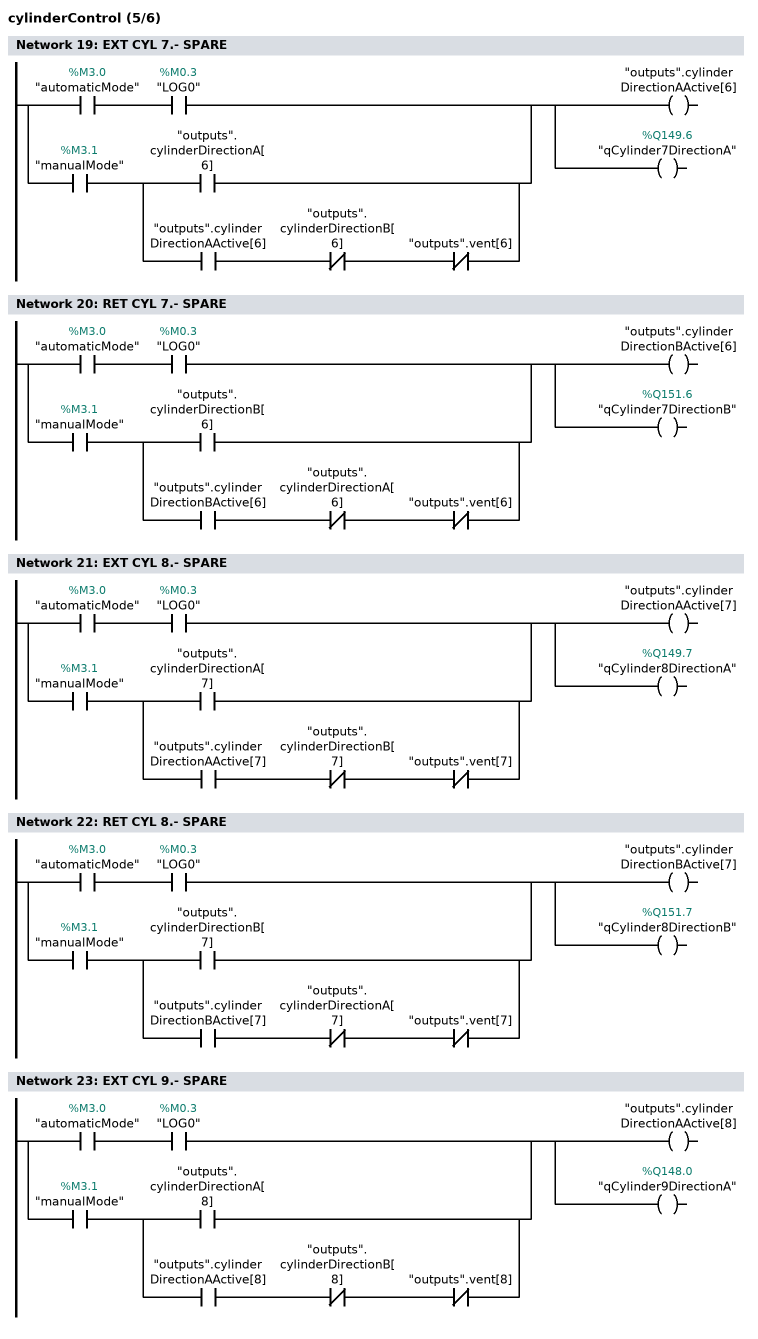
   RUNG wire#powerrail
      Contact( "automaticMode" )
      Contact( "LOG0" )
      wire#w1
      Coil( "outputs".cylinderDirectionAActive[6] )
   END_RUNG
   RUNG wire#powerrail
      Contact( "manualMode" )
      wire#w2
      Contact( "outputs".cylinderDirectionA[6] )
   END_RUNG wire#w1
   RUNG wire#w2
      Contact( "outputs".cylinderDirectionAActive[6] )
      I_Contact( "outputs".cylinderDirectionB[6] )
      I_Contact( "outputs".vent[6] )
   END_RUNG wire#w1
   RUNG wire#w1
      Coil( "qCylinder7DirectionA" )
   END_RUNG
   // the same network as SCL:
   #_w1 := ("automaticMode" AND "LOG0") OR ("manualMode" AND ("outputs".cylinderDirectionA[6] OR ("outputs".cylinderDirectionAActive[6] AND NOT "outputs".cylinderDirectionB[6] AND NOT "outputs".vent[6])));
   "outputs".cylinderDirectionAActive[6] := ("automaticMode" AND "LOG0") OR ("manualMode" AND ("outputs".cylinderDirectionA[6] OR ("outputs".cylinderDirectionAActive[6] AND NOT "outputs".cylinderDirectionB[6] AND NOT "outputs".vent[6])));
   "qCylinder7DirectionA" := #_w1;
END_REGION

REGION Network 20: RET CYL 7.- SPARE
   RUNG wire#powerrail
      Contact( "automaticMode" )
      Contact( "LOG0" )
      wire#w1
      Coil( "outputs".cylinderDirectionBActive[6] )
   END_RUNG
   RUNG wire#powerrail
      Contact( "manualMode" )
      wire#w2
      Contact( "outputs".cylinderDirectionB[6] )
   END_RUNG wire#w1
   RUNG wire#w2
      Contact( "outputs".cylinderDirectionBActive[6] )
      I_Contact( "outputs".cylinderDirectionA[6] )
      I_Contact( "outputs".vent[6] )
   END_RUNG wire#w1
   RUNG wire#w1
      Coil( "qCylinder7DirectionB" )
   END_RUNG
   // the same network as SCL:
   #_w1 := ("automaticMode" AND "LOG0") OR ("manualMode" AND ("outputs".cylinderDirectionB[6] OR ("outputs".cylinderDirectionBActive[6] AND NOT "outputs".cylinderDirectionA[6] AND NOT "outputs".vent[6])));
   "outputs".cylinderDirectionBActive[6] := ("automaticMode" AND "LOG0") OR ("manualMode" AND ("outputs".cylinderDirectionB[6] OR ("outputs".cylinderDirectionBActive[6] AND NOT "outputs".cylinderDirectionA[6] AND NOT "outputs".vent[6])));
   "qCylinder7DirectionB" := #_w1;
END_REGION

REGION Network 21: EXT CYL 8.- SPARE
   RUNG wire#powerrail
      Contact( "automaticMode" )
      Contact( "LOG0" )
      wire#w1
      Coil( "outputs".cylinderDirectionAActive[7] )
   END_RUNG
   RUNG wire#powerrail
      Contact( "manualMode" )
      wire#w2
      Contact( "outputs".cylinderDirectionA[7] )
   END_RUNG wire#w1
   RUNG wire#w2
      Contact( "outputs".cylinderDirectionAActive[7] )
      I_Contact( "outputs".cylinderDirectionB[7] )
      I_Contact( "outputs".vent[7] )
   END_RUNG wire#w1
   RUNG wire#w1
      Coil( "qCylinder8DirectionA" )
   END_RUNG
   // the same network as SCL:
   #_w1 := ("automaticMode" AND "LOG0") OR ("manualMode" AND ("outputs".cylinderDirectionA[7] OR ("outputs".cylinderDirectionAActive[7] AND NOT "outputs".cylinderDirectionB[7] AND NOT "outputs".vent[7])));
   "outputs".cylinderDirectionAActive[7] := ("automaticMode" AND "LOG0") OR ("manualMode" AND ("outputs".cylinderDirectionA[7] OR ("outputs".cylinderDirectionAActive[7] AND NOT "outputs".cylinderDirectionB[7] AND NOT "outputs".vent[7])));
   "qCylinder8DirectionA" := #_w1;
END_REGION

REGION Network 22: RET CYL 8.- SPARE
   RUNG wire#powerrail
      Contact( "automaticMode" )
      Contact( "LOG0" )
      wire#w1
      Coil( "outputs".cylinderDirectionBActive[7] )
   END_RUNG
   RUNG wire#powerrail
      Contact( "manualMode" )
      wire#w2
      Contact( "outputs".cylinderDirectionB[7] )
   END_RUNG wire#w1
   RUNG wire#w2
      Contact( "outputs".cylinderDirectionBActive[7] )
      I_Contact( "outputs".cylinderDirectionA[7] )
      I_Contact( "outputs".vent[7] )
   END_RUNG wire#w1
   RUNG wire#w1
      Coil( "qCylinder8DirectionB" )
   END_RUNG
   // the same network as SCL:
   #_w1 := ("automaticMode" AND "LOG0") OR ("manualMode" AND ("outputs".cylinderDirectionB[7] OR ("outputs".cylinderDirectionBActive[7] AND NOT "outputs".cylinderDirectionA[7] AND NOT "outputs".vent[7])));
   "outputs".cylinderDirectionBActive[7] := ("automaticMode" AND "LOG0") OR ("manualMode" AND ("outputs".cylinderDirectionB[7] OR ("outputs".cylinderDirectionBActive[7] AND NOT "outputs".cylinderDirectionA[7] AND NOT "outputs".vent[7])));
   "qCylinder8DirectionB" := #_w1;
END_REGION

REGION Network 23: EXT CYL 9.- SPARE
   RUNG wire#powerrail
      Contact( "automaticMode" )
      Contact( "LOG0" )
      wire#w1
      Coil( "outputs".cylinderDirectionAActive[8] )
   END_RUNG
   RUNG wire#powerrail
      Contact( "manualMode" )
      wire#w2
      Contact( "outputs".cylinderDirectionA[8] )
   END_RUNG wire#w1
   RUNG wire#w2
      Contact( "outputs".cylinderDirectionAActive[8] )
      I_Contact( "outputs".cylinderDirectionB[8] )
      I_Contact( "outputs".vent[8] )
   END_RUNG wire#w1
   RUNG wire#w1
      Coil( "qCylinder9DirectionA" )
   END_RUNG
   // the same network as SCL:
   #_w1 := ("automaticMode" AND "LOG0") OR ("manualMode" AND ("outputs".cylinderDirectionA[8] OR ("outputs".cylinderDirectionAActive[8] AND NOT "outputs".cylinderDirectionB[8] AND NOT "outputs".vent[8])));
   "outputs".cylinderDirectionAActive[8] := ("automaticMode" AND "LOG0") OR ("manualMode" AND ("outputs".cylinderDirectionA[8] OR ("outputs".cylinderDirectionAActive[8] AND NOT "outputs".cylinderDirectionB[8] AND NOT "outputs".vent[8])));
   "qCylinder9DirectionA" := #_w1;
END_REGION

REGION Network 24: RET CYL 9.- SPARE
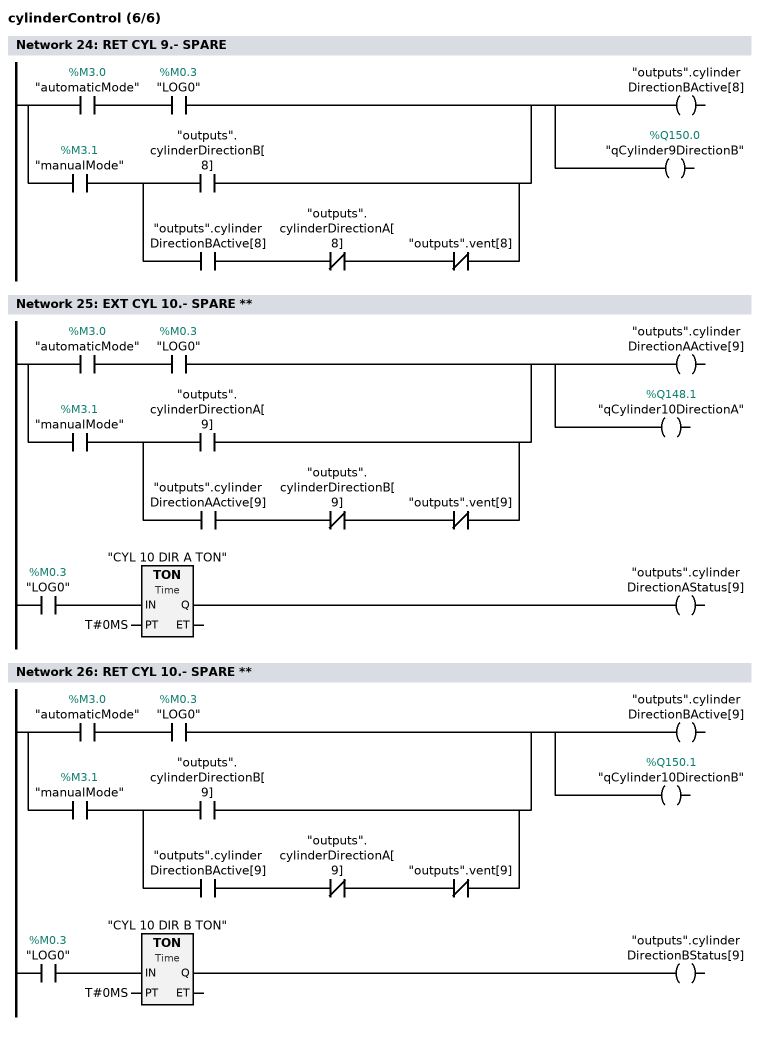
   RUNG wire#powerrail
      Contact( "automaticMode" )
      Contact( "LOG0" )
      wire#w1
      Coil( "outputs".cylinderDirectionBActive[8] )
   END_RUNG
   RUNG wire#powerrail
      Contact( "manualMode" )
      wire#w2
      Contact( "outputs".cylinderDirectionB[8] )
   END_RUNG wire#w1
   RUNG wire#w2
      Contact( "outputs".cylinderDirectionBActive[8] )
      I_Contact( "outputs".cylinderDirectionA[8] )
      I_Contact( "outputs".vent[8] )
   END_RUNG wire#w1
   RUNG wire#w1
      Coil( "qCylinder9DirectionB" )
   END_RUNG
   // the same network as SCL:
   #_w1 := ("automaticMode" AND "LOG0") OR ("manualMode" AND ("outputs".cylinderDirectionB[8] OR ("outputs".cylinderDirectionBActive[8] AND NOT "outputs".cylinderDirectionA[8] AND NOT "outputs".vent[8])));
   "outputs".cylinderDirectionBActive[8] := ("automaticMode" AND "LOG0") OR ("manualMode" AND ("outputs".cylinderDirectionB[8] OR ("outputs".cylinderDirectionBActive[8] AND NOT "outputs".cylinderDirectionA[8] AND NOT "outputs".vent[8])));
   "qCylinder9DirectionB" := #_w1;
END_REGION

REGION Network 25: EXT CYL 10.- SPARE **
   RUNG wire#powerrail
      Contact( "automaticMode" )
      Contact( "LOG0" )
      wire#w1
      Coil( "outputs".cylinderDirectionAActive[9] )
   END_RUNG
   RUNG wire#powerrail
      Contact( "manualMode" )
      wire#w2
      Contact( "outputs".cylinderDirectionA[9] )
   END_RUNG wire#w1
   RUNG wire#w2
      Contact( "outputs".cylinderDirectionAActive[9] )
      I_Contact( "outputs".cylinderDirectionB[9] )
      I_Contact( "outputs".vent[9] )
   END_RUNG wire#w1
   RUNG wire#w1
      Coil( "qCylinder10DirectionA" )
   END_RUNG
   RUNG wire#powerrail
      Contact( "LOG0" )
      { S7_Templates := "time_type := Time" } "CYL 10 DIR A TON".TON(pt := T#0MS, et =>)
      Coil( "outputs".cylinderDirectionAStatus[9] )
   END_RUNG
   // the same network as SCL:
   #_w1 := ("automaticMode" AND "LOG0") OR ("manualMode" AND ("outputs".cylinderDirectionA[9] OR ("outputs".cylinderDirectionAActive[9] AND NOT "outputs".cylinderDirectionB[9] AND NOT "outputs".vent[9])));
   "outputs".cylinderDirectionAActive[9] := ("automaticMode" AND "LOG0") OR ("manualMode" AND ("outputs".cylinderDirectionA[9] OR ("outputs".cylinderDirectionAActive[9] AND NOT "outputs".cylinderDirectionB[9] AND NOT "outputs".vent[9])));
   "qCylinder10DirectionA" := #_w1;
   "CYL 10 DIR A TON".TON(IN := "LOG0", PT := T#0MS);
   "outputs".cylinderDirectionAStatus[9] := "CYL 10 DIR A TON".Q;
END_REGION

REGION Network 26: RET CYL 10.- SPARE **
   RUNG wire#powerrail
      Contact( "automaticMode" )
      Contact( "LOG0" )
      wire#w1
      Coil( "outputs".cylinderDirectionBActive[9] )
   END_RUNG
   RUNG wire#powerrail
      Contact( "manualMode" )
      wire#w2
      Contact( "outputs".cylinderDirectionB[9] )
   END_RUNG wire#w1
   RUNG wire#w2
      Contact( "outputs".cylinderDirectionBActive[9] )
      I_Contact( "outputs".cylinderDirectionA[9] )
      I_Contact( "outputs".vent[9] )
   END_RUNG wire#w1
   RUNG wire#w1
      Coil( "qCylinder10DirectionB" )
   END_RUNG
   RUNG wire#powerrail
      Contact( "LOG0" )
      { S7_Templates := "time_type := Time" } "CYL 10 DIR B TON".TON(pt := T#0MS, et =>)
      Coil( "outputs".cylinderDirectionBStatus[9] )
   END_RUNG
   // the same network as SCL:
   #_w1 := ("automaticMode" AND "LOG0") OR ("manualMode" AND ("outputs".cylinderDirectionB[9] OR ("outputs".cylinderDirectionBActive[9] AND NOT "outputs".cylinderDirectionA[9] AND NOT "outputs".vent[9])));
   "outputs".cylinderDirectionBActive[9] := ("automaticMode" AND "LOG0") OR ("manualMode" AND ("outputs".cylinderDirectionB[9] OR ("outputs".cylinderDirectionBActive[9] AND NOT "outputs".cylinderDirectionA[9] AND NOT "outputs".vent[9])));
   "qCylinder10DirectionB" := #_w1;
   "CYL 10 DIR B TON".TON(IN := "LOG0", PT := T#0MS);
   "outputs".cylinderDirectionBStatus[9] := "CYL 10 DIR B TON".Q;
END_REGION
END_FUNCTION

FUNCTION "outputsMapping" : Void   // FC8, LAD
{ S7_Optimized_Access := 'TRUE' }
VERSION : 0.1
// stored: AutoNumber true, IsIECCheckEnabled false, SetENOAutomatically false, UDAEnableTagReadback false
BEGIN

REGION Network 1: STATION AIR ACTIVATION
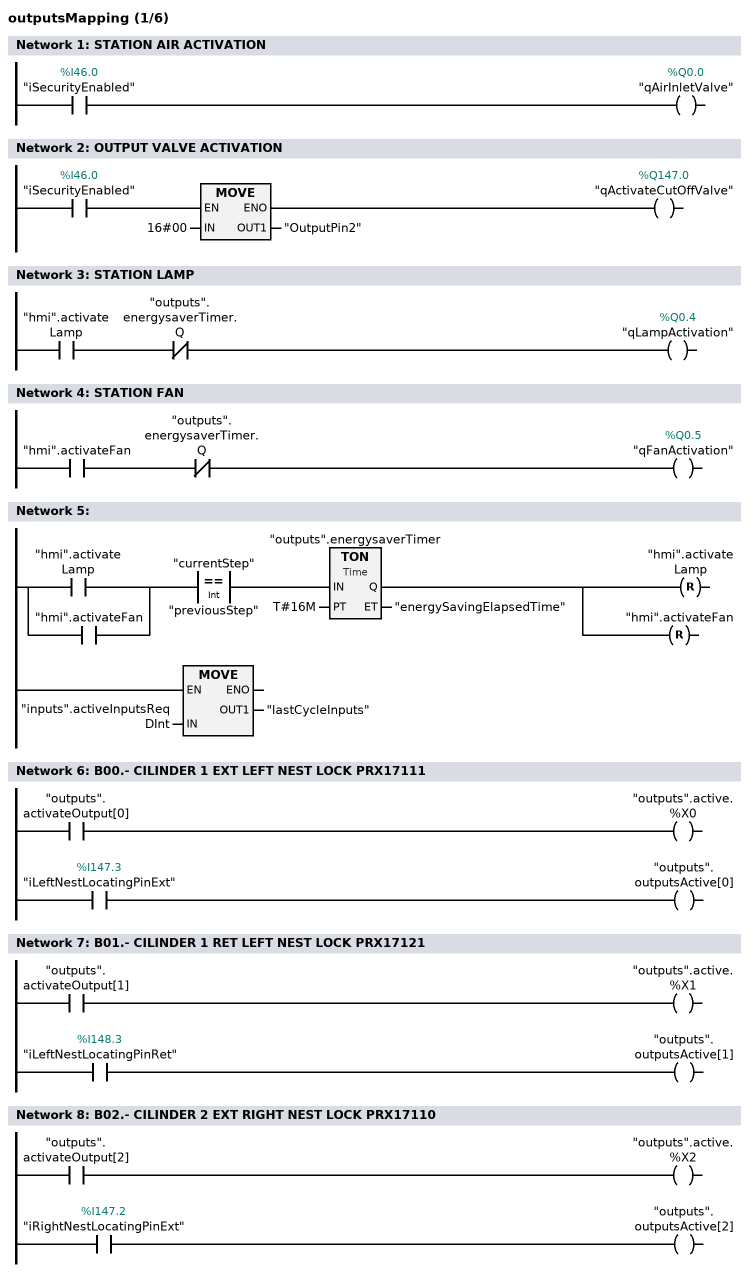
   RUNG wire#powerrail
      Contact( "iSecurityEnabled" )
      Coil( "qAirInletValve" )
   END_RUNG
   // the same network as SCL:
   "qAirInletValve" := "iSecurityEnabled";
END_REGION

REGION Network 2: OUTPUT VALVE ACTIVATION
   RUNG wire#powerrail
      Contact( "iSecurityEnabled" )
      Move(in := 16#00, out1 => "OutputPin2")
      Coil( "qActivateCutOffValve" )
   END_RUNG
   // the same network as SCL:
   IF "iSecurityEnabled" THEN "OutputPin2" := 16#00; END_IF;
   "qActivateCutOffValve" := "iSecurityEnabled";
END_REGION

REGION Network 3: STATION LAMP
   RUNG wire#powerrail
      Contact( "hmi".activateLamp )
      I_Contact( "outputs".energysaverTimer.Q )
      Coil( "qLampActivation" )
   END_RUNG
   // the same network as SCL:
   "qLampActivation" := "hmi".activateLamp AND NOT "outputs".energysaverTimer.Q;
END_REGION

REGION Network 4: STATION FAN
   RUNG wire#powerrail
      Contact( "hmi".activateFan )
      I_Contact( "outputs".energysaverTimer.Q )
      Coil( "qFanActivation" )
   END_RUNG
   // the same network as SCL:
   "qFanActivation" := "hmi".activateFan AND NOT "outputs".energysaverTimer.Q;
END_REGION

REGION Network 5
   RUNG wire#powerrail
      Contact( "hmi".activateLamp )
      wire#w1
      { S7_Templates := "SrcType := Int" } EQ_Contact(in1 := "currentStep", in2 := "previousStep")
      { S7_Templates := "time_type := Time" } "outputs".energysaverTimer.TON(pt := T#16M, et => "energySavingElapsedTime")
      wire#w2
      R_Coil( "hmi".activateLamp )
   END_RUNG
   RUNG wire#powerrail
      Contact( "hmi".activateFan )
   END_RUNG wire#w1
   RUNG wire#w2
      R_Coil( "hmi".activateFan )
   END_RUNG
   RUNG wire#powerrail
      Move(in := "inputs".activeInputsReqDInt, out1 => "lastCycleInputs")
   END_RUNG
   // the same network as SCL:
   "outputs".energysaverTimer.TON(IN := ("hmi".activateLamp OR "hmi".activateFan) AND ("currentStep" = "previousStep"),
                           PT := T#16M,
                           ET => "energySavingElapsedTime");
   IF "outputs".energysaverTimer.Q THEN
       "hmi".activateLamp := FALSE;
       "hmi".activateFan := FALSE;
   END_IF;
   "lastCycleInputs" := "inputs".activeInputsReqDInt;
END_REGION

REGION Network 6: B00.- CILINDER 1 EXT LEFT NEST LOCK PRX17111
   RUNG wire#powerrail
      Contact( "outputs".activateOutput[0] )
      Coil( "outputs".active.%X0 )
   END_RUNG
   RUNG wire#powerrail
      Contact( "iLeftNestLocatingPinExt" )
      Coil( "outputs".outputsActive[0] )
   END_RUNG
   // the same network as SCL:
   "outputs".active.%X0 := "outputs".activateOutput[0];
   "outputs".outputsActive[0] := "iLeftNestLocatingPinExt";
END_REGION

REGION Network 7: B01.- CILINDER 1 RET LEFT NEST LOCK PRX17121
   RUNG wire#powerrail
      Contact( "outputs".activateOutput[1] )
      Coil( "outputs".active.%X1 )
   END_RUNG
   RUNG wire#powerrail
      Contact( "iLeftNestLocatingPinRet" )
      Coil( "outputs".outputsActive[1] )
   END_RUNG
   // the same network as SCL:
   "outputs".active.%X1 := "outputs".activateOutput[1];
   "outputs".outputsActive[1] := "iLeftNestLocatingPinRet";
END_REGION

REGION Network 8: B02.- CILINDER 2 EXT RIGHT NEST LOCK PRX17110
   RUNG wire#powerrail
      Contact( "outputs".activateOutput[2] )
      Coil( "outputs".active.%X2 )
   END_RUNG
   RUNG wire#powerrail
      Contact( "iRightNestLocatingPinExt" )
      Coil( "outputs".outputsActive[2] )
   END_RUNG
   // the same network as SCL:
   "outputs".active.%X2 := "outputs".activateOutput[2];
   "outputs".outputsActive[2] := "iRightNestLocatingPinExt";
END_REGION

REGION Network 9: B03.- CILINDER 2 RET RIGHT NEST LOCK PRX17120
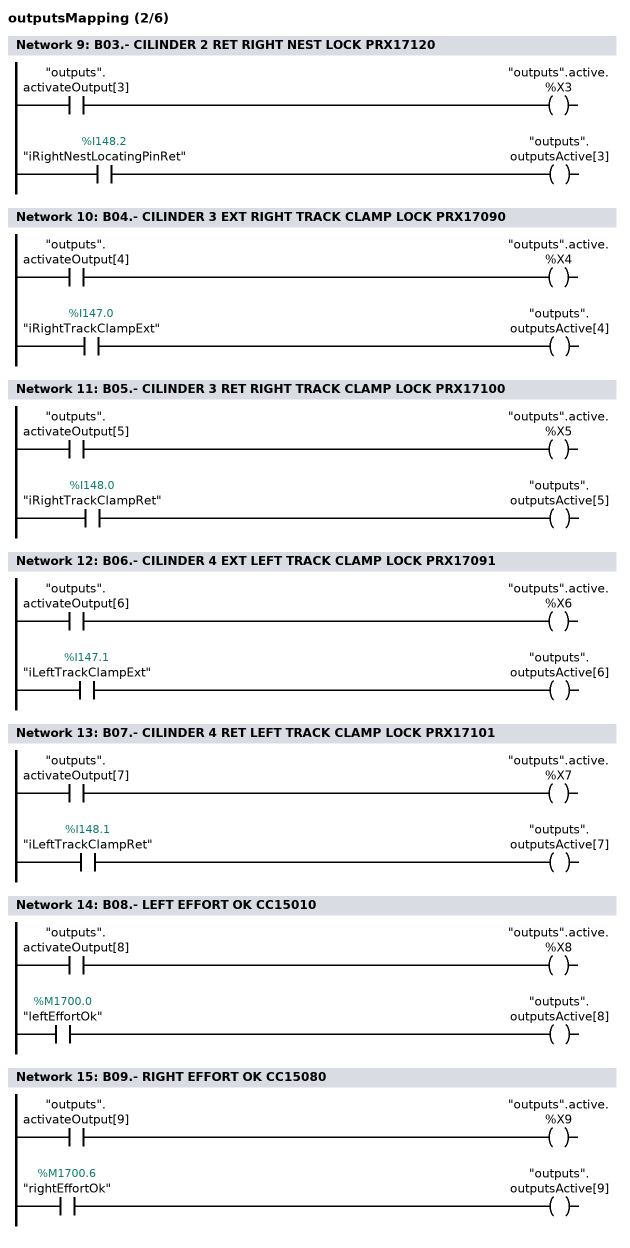
   RUNG wire#powerrail
      Contact( "outputs".activateOutput[3] )
      Coil( "outputs".active.%X3 )
   END_RUNG
   RUNG wire#powerrail
      Contact( "iRightNestLocatingPinRet" )
      Coil( "outputs".outputsActive[3] )
   END_RUNG
   // the same network as SCL:
   "outputs".active.%X3 := "outputs".activateOutput[3];
   "outputs".outputsActive[3] := "iRightNestLocatingPinRet";
END_REGION

REGION Network 10: B04.- CILINDER 3 EXT RIGHT TRACK CLAMP LOCK PRX17090
   RUNG wire#powerrail
      Contact( "outputs".activateOutput[4] )
      Coil( "outputs".active.%X4 )
   END_RUNG
   RUNG wire#powerrail
      Contact( "iRightTrackClampExt" )
      Coil( "outputs".outputsActive[4] )
   END_RUNG
   // the same network as SCL:
   "outputs".active.%X4 := "outputs".activateOutput[4];
   "outputs".outputsActive[4] := "iRightTrackClampExt";
END_REGION

REGION Network 11: B05.- CILINDER 3 RET RIGHT TRACK CLAMP LOCK PRX17100
   RUNG wire#powerrail
      Contact( "outputs".activateOutput[5] )
      Coil( "outputs".active.%X5 )
   END_RUNG
   RUNG wire#powerrail
      Contact( "iRightTrackClampRet" )
      Coil( "outputs".outputsActive[5] )
   END_RUNG
   // the same network as SCL:
   "outputs".active.%X5 := "outputs".activateOutput[5];
   "outputs".outputsActive[5] := "iRightTrackClampRet";
END_REGION

REGION Network 12: B06.- CILINDER 4 EXT LEFT TRACK CLAMP LOCK PRX17091
   RUNG wire#powerrail
      Contact( "outputs".activateOutput[6] )
      Coil( "outputs".active.%X6 )
   END_RUNG
   RUNG wire#powerrail
      Contact( "iLeftTrackClampExt" )
      Coil( "outputs".outputsActive[6] )
   END_RUNG
   // the same network as SCL:
   "outputs".active.%X6 := "outputs".activateOutput[6];
   "outputs".outputsActive[6] := "iLeftTrackClampExt";
END_REGION

REGION Network 13: B07.- CILINDER 4 RET LEFT TRACK CLAMP LOCK PRX17101
   RUNG wire#powerrail
      Contact( "outputs".activateOutput[7] )
      Coil( "outputs".active.%X7 )
   END_RUNG
   RUNG wire#powerrail
      Contact( "iLeftTrackClampRet" )
      Coil( "outputs".outputsActive[7] )
   END_RUNG
   // the same network as SCL:
   "outputs".active.%X7 := "outputs".activateOutput[7];
   "outputs".outputsActive[7] := "iLeftTrackClampRet";
END_REGION

REGION Network 14: B08.- LEFT EFFORT OK CC15010
   RUNG wire#powerrail
      Contact( "outputs".activateOutput[8] )
      Coil( "outputs".active.%X8 )
   END_RUNG
   RUNG wire#powerrail
      Contact( "leftEffortOk" )
      Coil( "outputs".outputsActive[8] )
   END_RUNG
   // the same network as SCL:
   "outputs".active.%X8 := "outputs".activateOutput[8];
   "outputs".outputsActive[8] := "leftEffortOk";
END_REGION

REGION Network 15: B09.- RIGHT EFFORT OK CC15080
   RUNG wire#powerrail
      Contact( "outputs".activateOutput[9] )
      Coil( "outputs".active.%X9 )
   END_RUNG
   RUNG wire#powerrail
      Contact( "rightEffortOk" )
      Coil( "outputs".outputsActive[9] )
   END_RUNG
   // the same network as SCL:
   "outputs".active.%X9 := "outputs".activateOutput[9];
   "outputs".outputsActive[9] := "rightEffortOk";
END_REGION

REGION Network 16: B10.- LEFT INSERTION OK DISTANCE SD14160
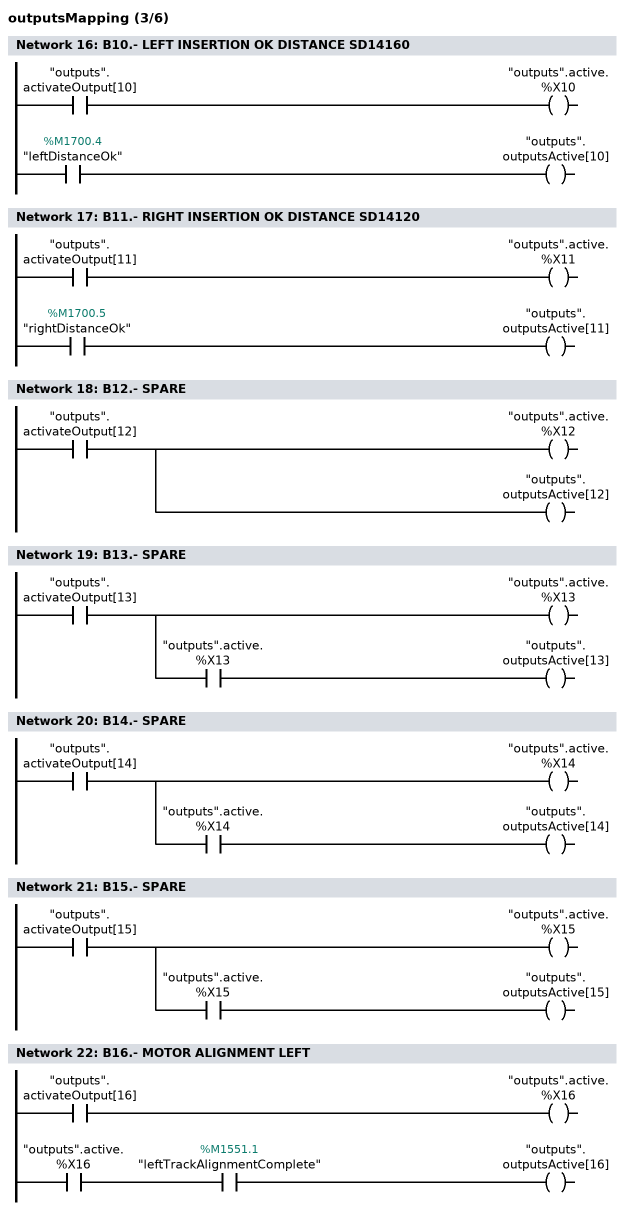
   RUNG wire#powerrail
      Contact( "outputs".activateOutput[10] )
      Coil( "outputs".active.%X10 )
   END_RUNG
   RUNG wire#powerrail
      Contact( "leftDistanceOk" )
      Coil( "outputs".outputsActive[10] )
   END_RUNG
   // the same network as SCL:
   "outputs".active.%X10 := "outputs".activateOutput[10];
   "outputs".outputsActive[10] := "leftDistanceOk";
END_REGION

REGION Network 17: B11.- RIGHT INSERTION OK DISTANCE SD14120
   RUNG wire#powerrail
      Contact( "outputs".activateOutput[11] )
      Coil( "outputs".active.%X11 )
   END_RUNG
   RUNG wire#powerrail
      Contact( "rightDistanceOk" )
      Coil( "outputs".outputsActive[11] )
   END_RUNG
   // the same network as SCL:
   "outputs".active.%X11 := "outputs".activateOutput[11];
   "outputs".outputsActive[11] := "rightDistanceOk";
END_REGION

REGION Network 18: B12.- SPARE
   RUNG wire#powerrail
      Contact( "outputs".activateOutput[12] )
      wire#w1
      Coil( "outputs".active.%X12 )
   END_RUNG
   RUNG wire#w1
      Coil( "outputs".outputsActive[12] )
   END_RUNG
   // the same network as SCL:
   "outputs".active.%X12 := "outputs".activateOutput[12];
   "outputs".outputsActive[12] := "outputs".activateOutput[12];
END_REGION

REGION Network 19: B13.- SPARE
   RUNG wire#powerrail
      Contact( "outputs".activateOutput[13] )
      wire#w1
      Coil( "outputs".active.%X13 )
   END_RUNG
   RUNG wire#w1
      Contact( "outputs".active.%X13 )
      Coil( "outputs".outputsActive[13] )
   END_RUNG
   // the same network as SCL:
   "outputs".active.%X13 := "outputs".activateOutput[13];
   "outputs".outputsActive[13] := "outputs".activateOutput[13] AND "outputs".active.%X13;
END_REGION

REGION Network 20: B14.- SPARE
   RUNG wire#powerrail
      Contact( "outputs".activateOutput[14] )
      wire#w1
      Coil( "outputs".active.%X14 )
   END_RUNG
   RUNG wire#w1
      Contact( "outputs".active.%X14 )
      Coil( "outputs".outputsActive[14] )
   END_RUNG
   // the same network as SCL:
   "outputs".active.%X14 := "outputs".activateOutput[14];
   "outputs".outputsActive[14] := "outputs".activateOutput[14] AND "outputs".active.%X14;
END_REGION

REGION Network 21: B15.- SPARE
   RUNG wire#powerrail
      Contact( "outputs".activateOutput[15] )
      wire#w1
      Coil( "outputs".active.%X15 )
   END_RUNG
   RUNG wire#w1
      Contact( "outputs".active.%X15 )
      Coil( "outputs".outputsActive[15] )
   END_RUNG
   // the same network as SCL:
   "outputs".active.%X15 := "outputs".activateOutput[15];
   "outputs".outputsActive[15] := "outputs".activateOutput[15] AND "outputs".active.%X15;
END_REGION

REGION Network 22: B16.- MOTOR ALIGNMENT LEFT
   RUNG wire#powerrail
      Contact( "outputs".activateOutput[16] )
      Coil( "outputs".active.%X16 )
   END_RUNG
   RUNG wire#powerrail
      Contact( "outputs".active.%X16 )
      Contact( "leftTrackAlignmentComplete" )
      Coil( "outputs".outputsActive[16] )
   END_RUNG
   // the same network as SCL:
   "outputs".active.%X16 := "outputs".activateOutput[16];
   "outputs".outputsActive[16] := "outputs".active.%X16 AND "leftTrackAlignmentComplete";
END_REGION

REGION Network 23: B17.- MOTOR ALIGNMENT RIGHT
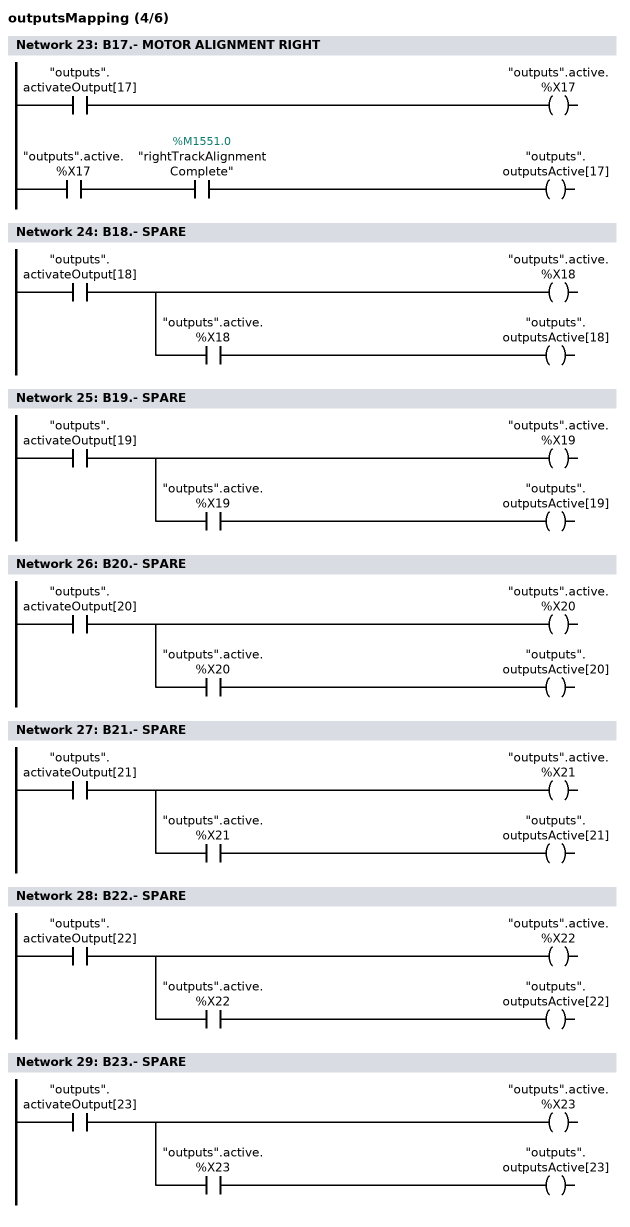
   RUNG wire#powerrail
      Contact( "outputs".activateOutput[17] )
      Coil( "outputs".active.%X17 )
   END_RUNG
   RUNG wire#powerrail
      Contact( "outputs".active.%X17 )
      Contact( "rightTrackAlignmentComplete" )
      Coil( "outputs".outputsActive[17] )
   END_RUNG
   // the same network as SCL:
   "outputs".active.%X17 := "outputs".activateOutput[17];
   "outputs".outputsActive[17] := "outputs".active.%X17 AND "rightTrackAlignmentComplete";
END_REGION

REGION Network 24: B18.- SPARE
   RUNG wire#powerrail
      Contact( "outputs".activateOutput[18] )
      wire#w1
      Coil( "outputs".active.%X18 )
   END_RUNG
   RUNG wire#w1
      Contact( "outputs".active.%X18 )
      Coil( "outputs".outputsActive[18] )
   END_RUNG
   // the same network as SCL:
   "outputs".active.%X18 := "outputs".activateOutput[18];
   "outputs".outputsActive[18] := "outputs".activateOutput[18] AND "outputs".active.%X18;
END_REGION

REGION Network 25: B19.- SPARE
   RUNG wire#powerrail
      Contact( "outputs".activateOutput[19] )
      wire#w1
      Coil( "outputs".active.%X19 )
   END_RUNG
   RUNG wire#w1
      Contact( "outputs".active.%X19 )
      Coil( "outputs".outputsActive[19] )
   END_RUNG
   // the same network as SCL:
   "outputs".active.%X19 := "outputs".activateOutput[19];
   "outputs".outputsActive[19] := "outputs".activateOutput[19] AND "outputs".active.%X19;
END_REGION

REGION Network 26: B20.- SPARE
   RUNG wire#powerrail
      Contact( "outputs".activateOutput[20] )
      wire#w1
      Coil( "outputs".active.%X20 )
   END_RUNG
   RUNG wire#w1
      Contact( "outputs".active.%X20 )
      Coil( "outputs".outputsActive[20] )
   END_RUNG
   // the same network as SCL:
   "outputs".active.%X20 := "outputs".activateOutput[20];
   "outputs".outputsActive[20] := "outputs".activateOutput[20] AND "outputs".active.%X20;
END_REGION

REGION Network 27: B21.- SPARE
   RUNG wire#powerrail
      Contact( "outputs".activateOutput[21] )
      wire#w1
      Coil( "outputs".active.%X21 )
   END_RUNG
   RUNG wire#w1
      Contact( "outputs".active.%X21 )
      Coil( "outputs".outputsActive[21] )
   END_RUNG
   // the same network as SCL:
   "outputs".active.%X21 := "outputs".activateOutput[21];
   "outputs".outputsActive[21] := "outputs".activateOutput[21] AND "outputs".active.%X21;
END_REGION

REGION Network 28: B22.- SPARE
   RUNG wire#powerrail
      Contact( "outputs".activateOutput[22] )
      wire#w1
      Coil( "outputs".active.%X22 )
   END_RUNG
   RUNG wire#w1
      Contact( "outputs".active.%X22 )
      Coil( "outputs".outputsActive[22] )
   END_RUNG
   // the same network as SCL:
   "outputs".active.%X22 := "outputs".activateOutput[22];
   "outputs".outputsActive[22] := "outputs".activateOutput[22] AND "outputs".active.%X22;
END_REGION

REGION Network 29: B23.- SPARE
   RUNG wire#powerrail
      Contact( "outputs".activateOutput[23] )
      wire#w1
      Coil( "outputs".active.%X23 )
   END_RUNG
   RUNG wire#w1
      Contact( "outputs".active.%X23 )
      Coil( "outputs".outputsActive[23] )
   END_RUNG
   // the same network as SCL:
   "outputs".active.%X23 := "outputs".activateOutput[23];
   "outputs".outputsActive[23] := "outputs".activateOutput[23] AND "outputs".active.%X23;
END_REGION

REGION Network 30: B24.- SPARE
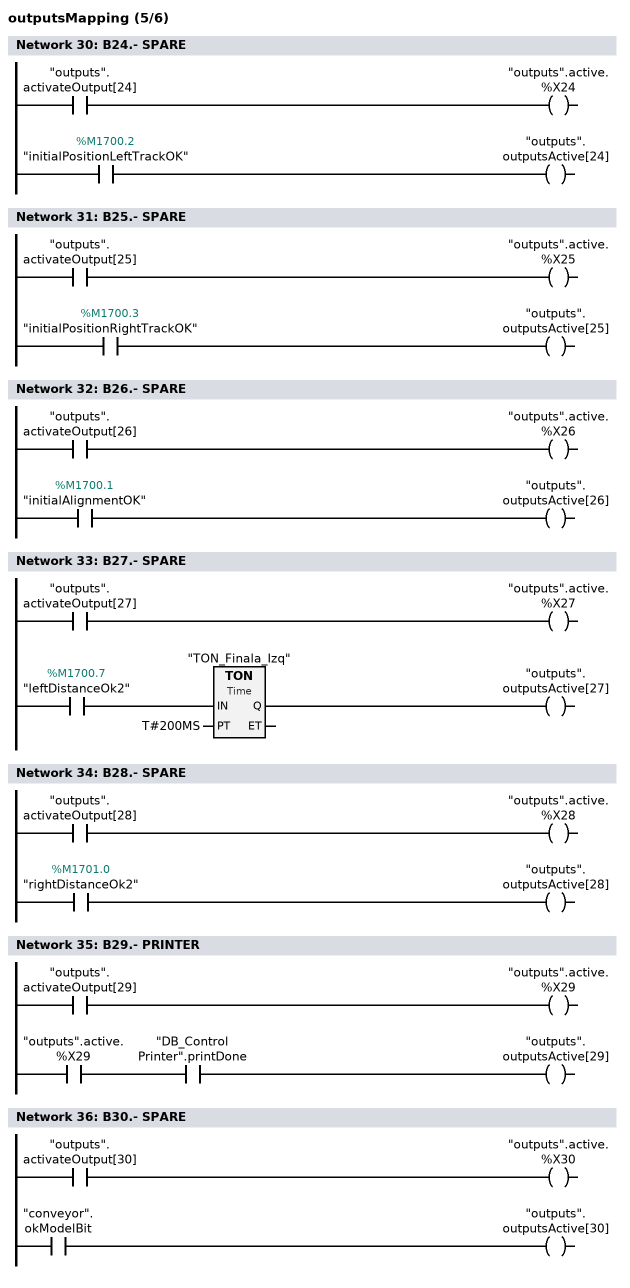
   RUNG wire#powerrail
      Contact( "outputs".activateOutput[24] )
      Coil( "outputs".active.%X24 )
   END_RUNG
   RUNG wire#powerrail
      Contact( "initialPositionLeftTrackOK" )
      Coil( "outputs".outputsActive[24] )
   END_RUNG
   // the same network as SCL:
   "outputs".active.%X24 := "outputs".activateOutput[24];
   "outputs".outputsActive[24] := "initialPositionLeftTrackOK";
END_REGION

REGION Network 31: B25.- SPARE
   RUNG wire#powerrail
      Contact( "outputs".activateOutput[25] )
      Coil( "outputs".active.%X25 )
   END_RUNG
   RUNG wire#powerrail
      Contact( "initialPositionRightTrackOK" )
      Coil( "outputs".outputsActive[25] )
   END_RUNG
   // the same network as SCL:
   "outputs".active.%X25 := "outputs".activateOutput[25];
   "outputs".outputsActive[25] := "initialPositionRightTrackOK";
END_REGION

REGION Network 32: B26.- SPARE
   RUNG wire#powerrail
      Contact( "outputs".activateOutput[26] )
      Coil( "outputs".active.%X26 )
   END_RUNG
   RUNG wire#powerrail
      Contact( "initialAlignmentOK" )
      Coil( "outputs".outputsActive[26] )
   END_RUNG
   // the same network as SCL:
   "outputs".active.%X26 := "outputs".activateOutput[26];
   "outputs".outputsActive[26] := "initialAlignmentOK";
END_REGION

REGION Network 33: B27.- SPARE
   RUNG wire#powerrail
      Contact( "outputs".activateOutput[27] )
      Coil( "outputs".active.%X27 )
   END_RUNG
   RUNG wire#powerrail
      Contact( "leftDistanceOk2" )
      { S7_Templates := "time_type := Time" } "TON_Finala_Izq".TON(pt := T#200MS, et =>)
      Coil( "outputs".outputsActive[27] )
   END_RUNG
   // the same network as SCL:
   "outputs".active.%X27 := "outputs".activateOutput[27];
   "TON_Finala_Izq".TON(IN := "leftDistanceOk2", PT := T#200MS);
   "outputs".outputsActive[27] := "TON_Finala_Izq".Q;
END_REGION

REGION Network 34: B28.- SPARE
   RUNG wire#powerrail
      Contact( "outputs".activateOutput[28] )
      Coil( "outputs".active.%X28 )
   END_RUNG
   RUNG wire#powerrail
      Contact( "rightDistanceOk2" )
      Coil( "outputs".outputsActive[28] )
   END_RUNG
   // the same network as SCL:
   "outputs".active.%X28 := "outputs".activateOutput[28];
   "outputs".outputsActive[28] := "rightDistanceOk2";
END_REGION

REGION Network 35: B29.- PRINTER
   RUNG wire#powerrail
      Contact( "outputs".activateOutput[29] )
      Coil( "outputs".active.%X29 )
   END_RUNG
   RUNG wire#powerrail
      Contact( "outputs".active.%X29 )
      Contact( "DB_ControlPrinter".printDone )
      Coil( "outputs".outputsActive[29] )
   END_RUNG
   // the same network as SCL:
   "outputs".active.%X29 := "outputs".activateOutput[29];
   "outputs".outputsActive[29] := "outputs".active.%X29 AND "DB_ControlPrinter".printDone;
END_REGION

REGION Network 36: B30.- SPARE
   RUNG wire#powerrail
      Contact( "outputs".activateOutput[30] )
      Coil( "outputs".active.%X30 )
   END_RUNG
   RUNG wire#powerrail
      Contact( "conveyor".okModelBit )
      Coil( "outputs".outputsActive[30] )
   END_RUNG
   // the same network as SCL:
   "outputs".active.%X30 := "outputs".activateOutput[30];
   "outputs".outputsActive[30] := "conveyor".okModelBit;
END_REGION

REGION Network 37: B31.- CYCLE TIME
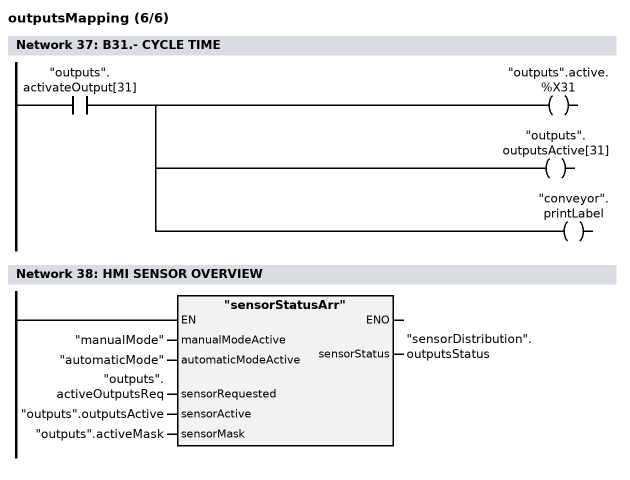
   RUNG wire#powerrail
      Contact( "outputs".activateOutput[31] )
      wire#w1
      Coil( "outputs".active.%X31 )
   END_RUNG
   RUNG wire#w1
      Coil( "outputs".outputsActive[31] )
   END_RUNG
   RUNG wire#w1
      Coil( "conveyor".printLabel )
   END_RUNG
   // the same network as SCL:
   "outputs".active.%X31 := "outputs".activateOutput[31];
   "outputs".outputsActive[31] := "outputs".activateOutput[31];
   "conveyor".printLabel := "outputs".activateOutput[31];
END_REGION

REGION Network 38: HMI SENSOR OVERVIEW
   RUNG wire#powerrail
      "sensorStatusArr"(manualModeActive := "manualMode", automaticModeActive := "automaticMode", sensorRequested := "outputs".activeOutputsReq, sensorActive := "outputs".outputsActive, sensorMask := "outputs".activeMask, sensorStatus => "sensorDistribution".outputsStatus)
   END_RUNG
   // the same network as SCL:
   "sensorStatusArr"(manualModeActive := "manualMode",
                     automaticModeActive := "automaticMode",
                     sensorRequested := "outputs".activeOutputsReq,
                     sensorActive := "outputs".outputsActive,
                     sensorMask := "outputs".activeMask,
                     sensorStatus => "sensorDistribution".outputsStatus);
END_REGION
END_FUNCTION

FUNCTION "sensorStatusArr" : Void   // FC38, LAD
{ S7_Optimized_Access := 'TRUE' }
VERSION : 0.1
// stored: AutoNumber true, IsIECCheckEnabled false, SetENOAutomatically false, UDAEnableTagReadback false
   VAR_INPUT
      manualModeActive : Bool;
      automaticModeActive : Bool;
      sensorRequested : Array[0..31] of Bool;
      sensorActive : Array[0..31] of Bool;
      sensorMask : Array[0..31] of Bool;
   END_VAR
   VAR_OUTPUT
      sensorStatus : Array[0..31] of Byte;
   END_VAR
BEGIN

REGION Network 1: Status 0
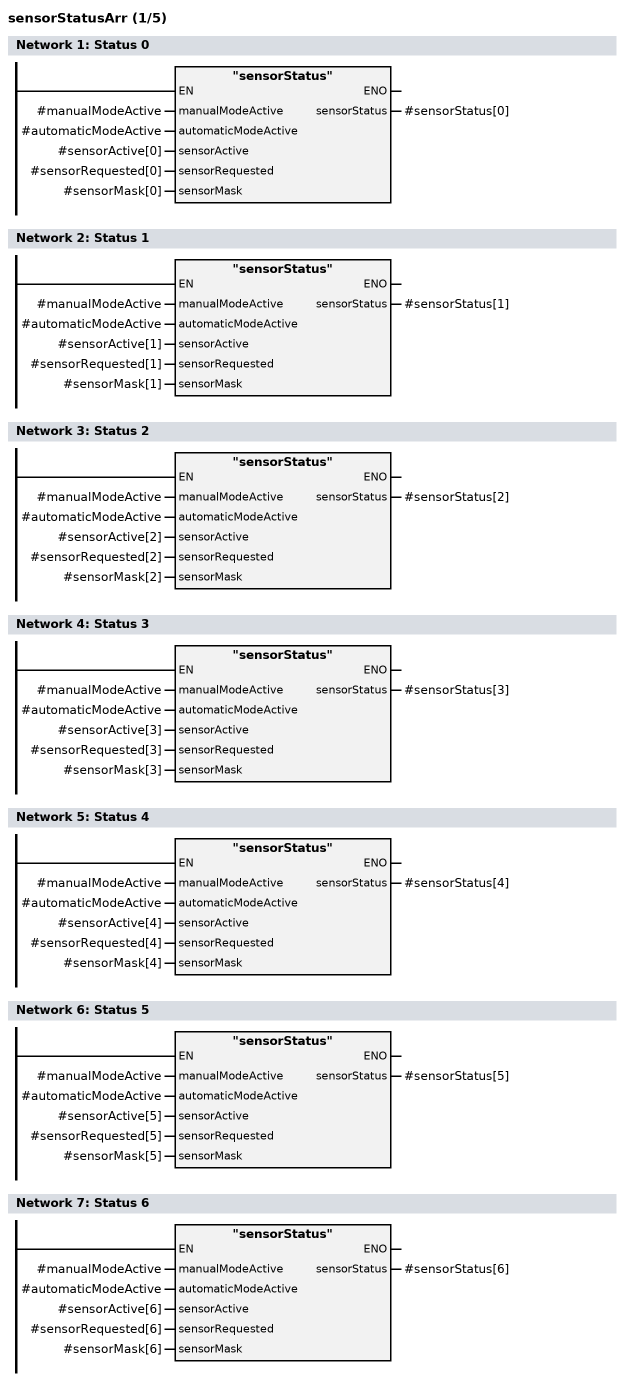
   RUNG wire#powerrail
      "sensorStatus"(manualModeActive := #manualModeActive, automaticModeActive := #automaticModeActive, sensorActive := #sensorActive[0], sensorRequested := #sensorRequested[0], sensorMask := #sensorMask[0], sensorStatus => #sensorStatus[0])
   END_RUNG
   // the same network as SCL:
   "sensorStatus"(manualModeActive := #manualModeActive,
                  automaticModeActive := #automaticModeActive,
                  sensorActive := #sensorActive[0],
                  sensorRequested := #sensorRequested[0],
                  sensorMask := #sensorMask[0],
                  sensorStatus => #sensorStatus[0]);
END_REGION

REGION Network 2: Status 1
   RUNG wire#powerrail
      "sensorStatus"(manualModeActive := #manualModeActive, automaticModeActive := #automaticModeActive, sensorActive := #sensorActive[1], sensorRequested := #sensorRequested[1], sensorMask := #sensorMask[1], sensorStatus => #sensorStatus[1])
   END_RUNG
   // the same network as SCL:
   "sensorStatus"(manualModeActive := #manualModeActive,
                  automaticModeActive := #automaticModeActive,
                  sensorActive := #sensorActive[1],
                  sensorRequested := #sensorRequested[1],
                  sensorMask := #sensorMask[1],
                  sensorStatus => #sensorStatus[1]);
END_REGION

REGION Network 3: Status 2
   RUNG wire#powerrail
      "sensorStatus"(manualModeActive := #manualModeActive, automaticModeActive := #automaticModeActive, sensorActive := #sensorActive[2], sensorRequested := #sensorRequested[2], sensorMask := #sensorMask[2], sensorStatus => #sensorStatus[2])
   END_RUNG
   // the same network as SCL:
   "sensorStatus"(manualModeActive := #manualModeActive,
                  automaticModeActive := #automaticModeActive,
                  sensorActive := #sensorActive[2],
                  sensorRequested := #sensorRequested[2],
                  sensorMask := #sensorMask[2],
                  sensorStatus => #sensorStatus[2]);
END_REGION

REGION Network 4: Status 3
   RUNG wire#powerrail
      "sensorStatus"(manualModeActive := #manualModeActive, automaticModeActive := #automaticModeActive, sensorActive := #sensorActive[3], sensorRequested := #sensorRequested[3], sensorMask := #sensorMask[3], sensorStatus => #sensorStatus[3])
   END_RUNG
   // the same network as SCL:
   "sensorStatus"(manualModeActive := #manualModeActive,
                  automaticModeActive := #automaticModeActive,
                  sensorActive := #sensorActive[3],
                  sensorRequested := #sensorRequested[3],
                  sensorMask := #sensorMask[3],
                  sensorStatus => #sensorStatus[3]);
END_REGION

REGION Network 5: Status 4
   RUNG wire#powerrail
      "sensorStatus"(manualModeActive := #manualModeActive, automaticModeActive := #automaticModeActive, sensorActive := #sensorActive[4], sensorRequested := #sensorRequested[4], sensorMask := #sensorMask[4], sensorStatus => #sensorStatus[4])
   END_RUNG
   // the same network as SCL:
   "sensorStatus"(manualModeActive := #manualModeActive,
                  automaticModeActive := #automaticModeActive,
                  sensorActive := #sensorActive[4],
                  sensorRequested := #sensorRequested[4],
                  sensorMask := #sensorMask[4],
                  sensorStatus => #sensorStatus[4]);
END_REGION

REGION Network 6: Status 5
   RUNG wire#powerrail
      "sensorStatus"(manualModeActive := #manualModeActive, automaticModeActive := #automaticModeActive, sensorActive := #sensorActive[5], sensorRequested := #sensorRequested[5], sensorMask := #sensorMask[5], sensorStatus => #sensorStatus[5])
   END_RUNG
   // the same network as SCL:
   "sensorStatus"(manualModeActive := #manualModeActive,
                  automaticModeActive := #automaticModeActive,
                  sensorActive := #sensorActive[5],
                  sensorRequested := #sensorRequested[5],
                  sensorMask := #sensorMask[5],
                  sensorStatus => #sensorStatus[5]);
END_REGION

REGION Network 7: Status 6
   RUNG wire#powerrail
      "sensorStatus"(manualModeActive := #manualModeActive, automaticModeActive := #automaticModeActive, sensorActive := #sensorActive[6], sensorRequested := #sensorRequested[6], sensorMask := #sensorMask[6], sensorStatus => #sensorStatus[6])
   END_RUNG
   // the same network as SCL:
   "sensorStatus"(manualModeActive := #manualModeActive,
                  automaticModeActive := #automaticModeActive,
                  sensorActive := #sensorActive[6],
                  sensorRequested := #sensorRequested[6],
                  sensorMask := #sensorMask[6],
                  sensorStatus => #sensorStatus[6]);
END_REGION

REGION Network 8: Status 7
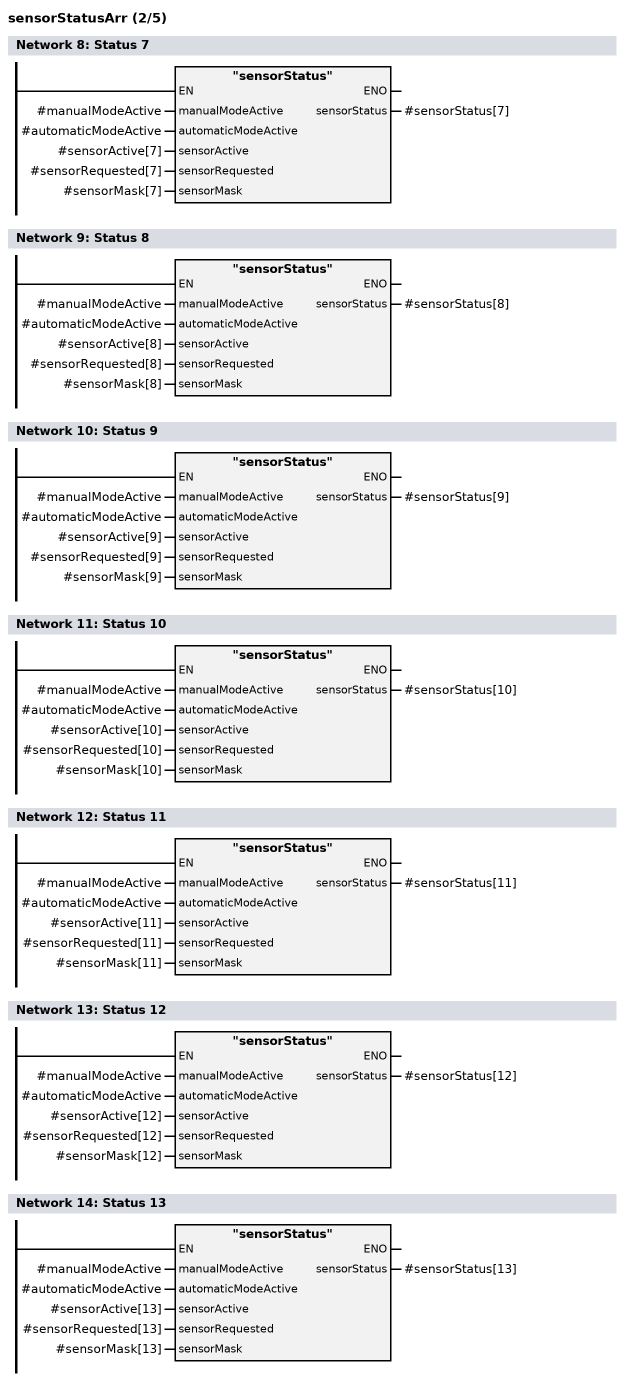
   RUNG wire#powerrail
      "sensorStatus"(manualModeActive := #manualModeActive, automaticModeActive := #automaticModeActive, sensorActive := #sensorActive[7], sensorRequested := #sensorRequested[7], sensorMask := #sensorMask[7], sensorStatus => #sensorStatus[7])
   END_RUNG
   // the same network as SCL:
   "sensorStatus"(manualModeActive := #manualModeActive,
                  automaticModeActive := #automaticModeActive,
                  sensorActive := #sensorActive[7],
                  sensorRequested := #sensorRequested[7],
                  sensorMask := #sensorMask[7],
                  sensorStatus => #sensorStatus[7]);
END_REGION

REGION Network 9: Status 8
   RUNG wire#powerrail
      "sensorStatus"(manualModeActive := #manualModeActive, automaticModeActive := #automaticModeActive, sensorActive := #sensorActive[8], sensorRequested := #sensorRequested[8], sensorMask := #sensorMask[8], sensorStatus => #sensorStatus[8])
   END_RUNG
   // the same network as SCL:
   "sensorStatus"(manualModeActive := #manualModeActive,
                  automaticModeActive := #automaticModeActive,
                  sensorActive := #sensorActive[8],
                  sensorRequested := #sensorRequested[8],
                  sensorMask := #sensorMask[8],
                  sensorStatus => #sensorStatus[8]);
END_REGION

REGION Network 10: Status 9
   RUNG wire#powerrail
      "sensorStatus"(manualModeActive := #manualModeActive, automaticModeActive := #automaticModeActive, sensorActive := #sensorActive[9], sensorRequested := #sensorRequested[9], sensorMask := #sensorMask[9], sensorStatus => #sensorStatus[9])
   END_RUNG
   // the same network as SCL:
   "sensorStatus"(manualModeActive := #manualModeActive,
                  automaticModeActive := #automaticModeActive,
                  sensorActive := #sensorActive[9],
                  sensorRequested := #sensorRequested[9],
                  sensorMask := #sensorMask[9],
                  sensorStatus => #sensorStatus[9]);
END_REGION

REGION Network 11: Status 10
   RUNG wire#powerrail
      "sensorStatus"(manualModeActive := #manualModeActive, automaticModeActive := #automaticModeActive, sensorActive := #sensorActive[10], sensorRequested := #sensorRequested[10], sensorMask := #sensorMask[10], sensorStatus => #sensorStatus[10])
   END_RUNG
   // the same network as SCL:
   "sensorStatus"(manualModeActive := #manualModeActive,
                  automaticModeActive := #automaticModeActive,
                  sensorActive := #sensorActive[10],
                  sensorRequested := #sensorRequested[10],
                  sensorMask := #sensorMask[10],
                  sensorStatus => #sensorStatus[10]);
END_REGION

REGION Network 12: Status 11
   RUNG wire#powerrail
      "sensorStatus"(manualModeActive := #manualModeActive, automaticModeActive := #automaticModeActive, sensorActive := #sensorActive[11], sensorRequested := #sensorRequested[11], sensorMask := #sensorMask[11], sensorStatus => #sensorStatus[11])
   END_RUNG
   // the same network as SCL:
   "sensorStatus"(manualModeActive := #manualModeActive,
                  automaticModeActive := #automaticModeActive,
                  sensorActive := #sensorActive[11],
                  sensorRequested := #sensorRequested[11],
                  sensorMask := #sensorMask[11],
                  sensorStatus => #sensorStatus[11]);
END_REGION

REGION Network 13: Status 12
   RUNG wire#powerrail
      "sensorStatus"(manualModeActive := #manualModeActive, automaticModeActive := #automaticModeActive, sensorActive := #sensorActive[12], sensorRequested := #sensorRequested[12], sensorMask := #sensorMask[12], sensorStatus => #sensorStatus[12])
   END_RUNG
   // the same network as SCL:
   "sensorStatus"(manualModeActive := #manualModeActive,
                  automaticModeActive := #automaticModeActive,
                  sensorActive := #sensorActive[12],
                  sensorRequested := #sensorRequested[12],
                  sensorMask := #sensorMask[12],
                  sensorStatus => #sensorStatus[12]);
END_REGION

REGION Network 14: Status 13
   RUNG wire#powerrail
      "sensorStatus"(manualModeActive := #manualModeActive, automaticModeActive := #automaticModeActive, sensorActive := #sensorActive[13], sensorRequested := #sensorRequested[13], sensorMask := #sensorMask[13], sensorStatus => #sensorStatus[13])
   END_RUNG
   // the same network as SCL:
   "sensorStatus"(manualModeActive := #manualModeActive,
                  automaticModeActive := #automaticModeActive,
                  sensorActive := #sensorActive[13],
                  sensorRequested := #sensorRequested[13],
                  sensorMask := #sensorMask[13],
                  sensorStatus => #sensorStatus[13]);
END_REGION

REGION Network 15: Status 14
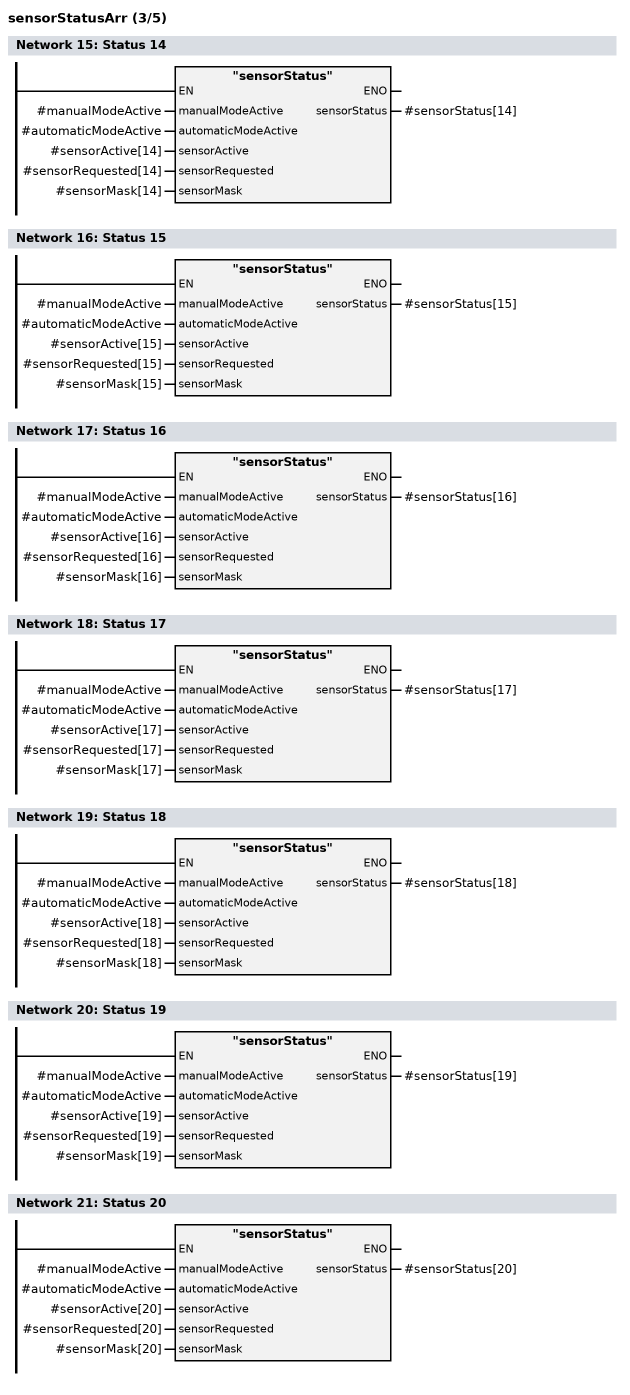
   RUNG wire#powerrail
      "sensorStatus"(manualModeActive := #manualModeActive, automaticModeActive := #automaticModeActive, sensorActive := #sensorActive[14], sensorRequested := #sensorRequested[14], sensorMask := #sensorMask[14], sensorStatus => #sensorStatus[14])
   END_RUNG
   // the same network as SCL:
   "sensorStatus"(manualModeActive := #manualModeActive,
                  automaticModeActive := #automaticModeActive,
                  sensorActive := #sensorActive[14],
                  sensorRequested := #sensorRequested[14],
                  sensorMask := #sensorMask[14],
                  sensorStatus => #sensorStatus[14]);
END_REGION

REGION Network 16: Status 15
   RUNG wire#powerrail
      "sensorStatus"(manualModeActive := #manualModeActive, automaticModeActive := #automaticModeActive, sensorActive := #sensorActive[15], sensorRequested := #sensorRequested[15], sensorMask := #sensorMask[15], sensorStatus => #sensorStatus[15])
   END_RUNG
   // the same network as SCL:
   "sensorStatus"(manualModeActive := #manualModeActive,
                  automaticModeActive := #automaticModeActive,
                  sensorActive := #sensorActive[15],
                  sensorRequested := #sensorRequested[15],
                  sensorMask := #sensorMask[15],
                  sensorStatus => #sensorStatus[15]);
END_REGION

REGION Network 17: Status 16
   RUNG wire#powerrail
      "sensorStatus"(manualModeActive := #manualModeActive, automaticModeActive := #automaticModeActive, sensorActive := #sensorActive[16], sensorRequested := #sensorRequested[16], sensorMask := #sensorMask[16], sensorStatus => #sensorStatus[16])
   END_RUNG
   // the same network as SCL:
   "sensorStatus"(manualModeActive := #manualModeActive,
                  automaticModeActive := #automaticModeActive,
                  sensorActive := #sensorActive[16],
                  sensorRequested := #sensorRequested[16],
                  sensorMask := #sensorMask[16],
                  sensorStatus => #sensorStatus[16]);
END_REGION

REGION Network 18: Status 17
   RUNG wire#powerrail
      "sensorStatus"(manualModeActive := #manualModeActive, automaticModeActive := #automaticModeActive, sensorActive := #sensorActive[17], sensorRequested := #sensorRequested[17], sensorMask := #sensorMask[17], sensorStatus => #sensorStatus[17])
   END_RUNG
   // the same network as SCL:
   "sensorStatus"(manualModeActive := #manualModeActive,
                  automaticModeActive := #automaticModeActive,
                  sensorActive := #sensorActive[17],
                  sensorRequested := #sensorRequested[17],
                  sensorMask := #sensorMask[17],
                  sensorStatus => #sensorStatus[17]);
END_REGION

REGION Network 19: Status 18
   RUNG wire#powerrail
      "sensorStatus"(manualModeActive := #manualModeActive, automaticModeActive := #automaticModeActive, sensorActive := #sensorActive[18], sensorRequested := #sensorRequested[18], sensorMask := #sensorMask[18], sensorStatus => #sensorStatus[18])
   END_RUNG
   // the same network as SCL:
   "sensorStatus"(manualModeActive := #manualModeActive,
                  automaticModeActive := #automaticModeActive,
                  sensorActive := #sensorActive[18],
                  sensorRequested := #sensorRequested[18],
                  sensorMask := #sensorMask[18],
                  sensorStatus => #sensorStatus[18]);
END_REGION

REGION Network 20: Status 19
   RUNG wire#powerrail
      "sensorStatus"(manualModeActive := #manualModeActive, automaticModeActive := #automaticModeActive, sensorActive := #sensorActive[19], sensorRequested := #sensorRequested[19], sensorMask := #sensorMask[19], sensorStatus => #sensorStatus[19])
   END_RUNG
   // the same network as SCL:
   "sensorStatus"(manualModeActive := #manualModeActive,
                  automaticModeActive := #automaticModeActive,
                  sensorActive := #sensorActive[19],
                  sensorRequested := #sensorRequested[19],
                  sensorMask := #sensorMask[19],
                  sensorStatus => #sensorStatus[19]);
END_REGION

REGION Network 21: Status 20
   RUNG wire#powerrail
      "sensorStatus"(manualModeActive := #manualModeActive, automaticModeActive := #automaticModeActive, sensorActive := #sensorActive[20], sensorRequested := #sensorRequested[20], sensorMask := #sensorMask[20], sensorStatus => #sensorStatus[20])
   END_RUNG
   // the same network as SCL:
   "sensorStatus"(manualModeActive := #manualModeActive,
                  automaticModeActive := #automaticModeActive,
                  sensorActive := #sensorActive[20],
                  sensorRequested := #sensorRequested[20],
                  sensorMask := #sensorMask[20],
                  sensorStatus => #sensorStatus[20]);
END_REGION

REGION Network 22: Status 21
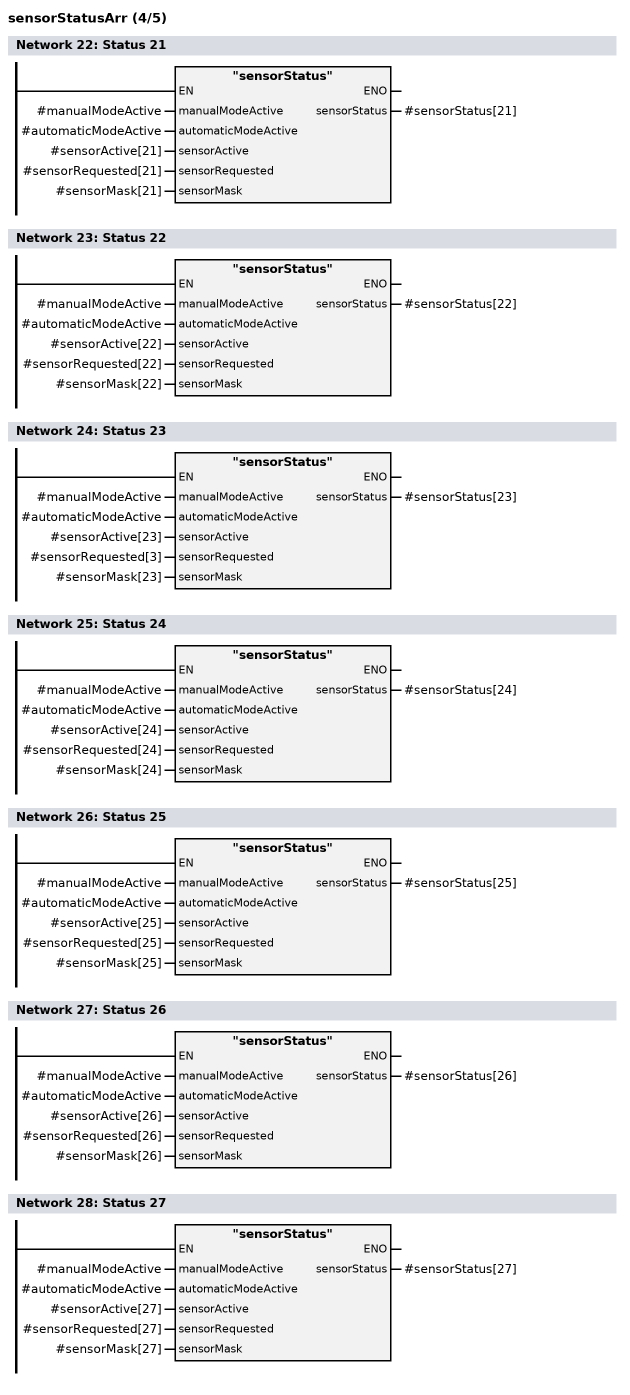
   RUNG wire#powerrail
      "sensorStatus"(manualModeActive := #manualModeActive, automaticModeActive := #automaticModeActive, sensorActive := #sensorActive[21], sensorRequested := #sensorRequested[21], sensorMask := #sensorMask[21], sensorStatus => #sensorStatus[21])
   END_RUNG
   // the same network as SCL:
   "sensorStatus"(manualModeActive := #manualModeActive,
                  automaticModeActive := #automaticModeActive,
                  sensorActive := #sensorActive[21],
                  sensorRequested := #sensorRequested[21],
                  sensorMask := #sensorMask[21],
                  sensorStatus => #sensorStatus[21]);
END_REGION

REGION Network 23: Status 22
   RUNG wire#powerrail
      "sensorStatus"(manualModeActive := #manualModeActive, automaticModeActive := #automaticModeActive, sensorActive := #sensorActive[22], sensorRequested := #sensorRequested[22], sensorMask := #sensorMask[22], sensorStatus => #sensorStatus[22])
   END_RUNG
   // the same network as SCL:
   "sensorStatus"(manualModeActive := #manualModeActive,
                  automaticModeActive := #automaticModeActive,
                  sensorActive := #sensorActive[22],
                  sensorRequested := #sensorRequested[22],
                  sensorMask := #sensorMask[22],
                  sensorStatus => #sensorStatus[22]);
END_REGION

REGION Network 24: Status 23
   RUNG wire#powerrail
      "sensorStatus"(manualModeActive := #manualModeActive, automaticModeActive := #automaticModeActive, sensorActive := #sensorActive[23], sensorRequested := #sensorRequested[3], sensorMask := #sensorMask[23], sensorStatus => #sensorStatus[23])
   END_RUNG
   // the same network as SCL:
   "sensorStatus"(manualModeActive := #manualModeActive,
                  automaticModeActive := #automaticModeActive,
                  sensorActive := #sensorActive[23],
                  sensorRequested := #sensorRequested[3],
                  sensorMask := #sensorMask[23],
                  sensorStatus => #sensorStatus[23]);
END_REGION

REGION Network 25: Status 24
   RUNG wire#powerrail
      "sensorStatus"(manualModeActive := #manualModeActive, automaticModeActive := #automaticModeActive, sensorActive := #sensorActive[24], sensorRequested := #sensorRequested[24], sensorMask := #sensorMask[24], sensorStatus => #sensorStatus[24])
   END_RUNG
   // the same network as SCL:
   "sensorStatus"(manualModeActive := #manualModeActive,
                  automaticModeActive := #automaticModeActive,
                  sensorActive := #sensorActive[24],
                  sensorRequested := #sensorRequested[24],
                  sensorMask := #sensorMask[24],
                  sensorStatus => #sensorStatus[24]);
END_REGION

REGION Network 26: Status 25
   RUNG wire#powerrail
      "sensorStatus"(manualModeActive := #manualModeActive, automaticModeActive := #automaticModeActive, sensorActive := #sensorActive[25], sensorRequested := #sensorRequested[25], sensorMask := #sensorMask[25], sensorStatus => #sensorStatus[25])
   END_RUNG
   // the same network as SCL:
   "sensorStatus"(manualModeActive := #manualModeActive,
                  automaticModeActive := #automaticModeActive,
                  sensorActive := #sensorActive[25],
                  sensorRequested := #sensorRequested[25],
                  sensorMask := #sensorMask[25],
                  sensorStatus => #sensorStatus[25]);
END_REGION

REGION Network 27: Status 26
   RUNG wire#powerrail
      "sensorStatus"(manualModeActive := #manualModeActive, automaticModeActive := #automaticModeActive, sensorActive := #sensorActive[26], sensorRequested := #sensorRequested[26], sensorMask := #sensorMask[26], sensorStatus => #sensorStatus[26])
   END_RUNG
   // the same network as SCL:
   "sensorStatus"(manualModeActive := #manualModeActive,
                  automaticModeActive := #automaticModeActive,
                  sensorActive := #sensorActive[26],
                  sensorRequested := #sensorRequested[26],
                  sensorMask := #sensorMask[26],
                  sensorStatus => #sensorStatus[26]);
END_REGION

REGION Network 28: Status 27
   RUNG wire#powerrail
      "sensorStatus"(manualModeActive := #manualModeActive, automaticModeActive := #automaticModeActive, sensorActive := #sensorActive[27], sensorRequested := #sensorRequested[27], sensorMask := #sensorMask[27], sensorStatus => #sensorStatus[27])
   END_RUNG
   // the same network as SCL:
   "sensorStatus"(manualModeActive := #manualModeActive,
                  automaticModeActive := #automaticModeActive,
                  sensorActive := #sensorActive[27],
                  sensorRequested := #sensorRequested[27],
                  sensorMask := #sensorMask[27],
                  sensorStatus => #sensorStatus[27]);
END_REGION

REGION Network 29: Status 28
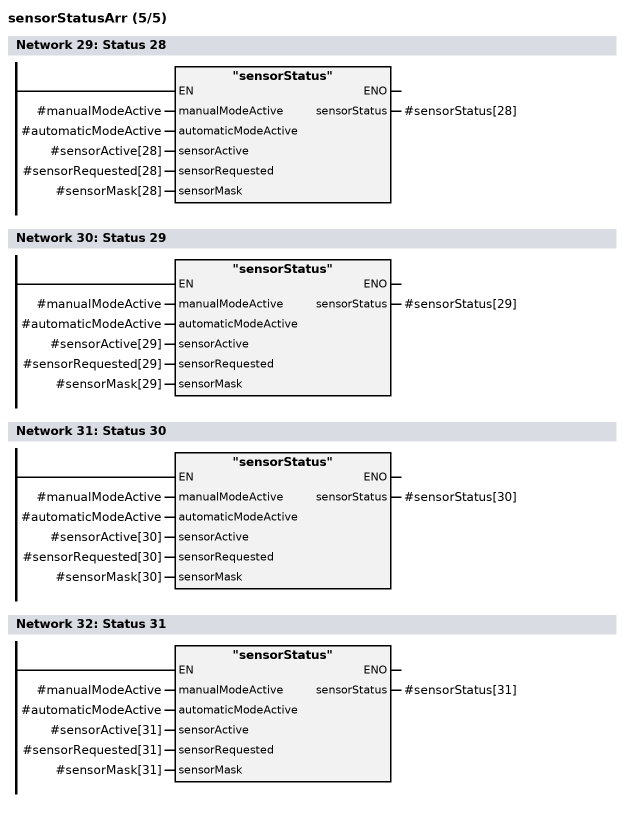
   RUNG wire#powerrail
      "sensorStatus"(manualModeActive := #manualModeActive, automaticModeActive := #automaticModeActive, sensorActive := #sensorActive[28], sensorRequested := #sensorRequested[28], sensorMask := #sensorMask[28], sensorStatus => #sensorStatus[28])
   END_RUNG
   // the same network as SCL:
   "sensorStatus"(manualModeActive := #manualModeActive,
                  automaticModeActive := #automaticModeActive,
                  sensorActive := #sensorActive[28],
                  sensorRequested := #sensorRequested[28],
                  sensorMask := #sensorMask[28],
                  sensorStatus => #sensorStatus[28]);
END_REGION

REGION Network 30: Status 29
   RUNG wire#powerrail
      "sensorStatus"(manualModeActive := #manualModeActive, automaticModeActive := #automaticModeActive, sensorActive := #sensorActive[29], sensorRequested := #sensorRequested[29], sensorMask := #sensorMask[29], sensorStatus => #sensorStatus[29])
   END_RUNG
   // the same network as SCL:
   "sensorStatus"(manualModeActive := #manualModeActive,
                  automaticModeActive := #automaticModeActive,
                  sensorActive := #sensorActive[29],
                  sensorRequested := #sensorRequested[29],
                  sensorMask := #sensorMask[29],
                  sensorStatus => #sensorStatus[29]);
END_REGION

REGION Network 31: Status 30
   RUNG wire#powerrail
      "sensorStatus"(manualModeActive := #manualModeActive, automaticModeActive := #automaticModeActive, sensorActive := #sensorActive[30], sensorRequested := #sensorRequested[30], sensorMask := #sensorMask[30], sensorStatus => #sensorStatus[30])
   END_RUNG
   // the same network as SCL:
   "sensorStatus"(manualModeActive := #manualModeActive,
                  automaticModeActive := #automaticModeActive,
                  sensorActive := #sensorActive[30],
                  sensorRequested := #sensorRequested[30],
                  sensorMask := #sensorMask[30],
                  sensorStatus => #sensorStatus[30]);
END_REGION

REGION Network 32: Status 31
   RUNG wire#powerrail
      "sensorStatus"(manualModeActive := #manualModeActive, automaticModeActive := #automaticModeActive, sensorActive := #sensorActive[31], sensorRequested := #sensorRequested[31], sensorMask := #sensorMask[31], sensorStatus => #sensorStatus[31])
   END_RUNG
   // the same network as SCL:
   "sensorStatus"(manualModeActive := #manualModeActive,
                  automaticModeActive := #automaticModeActive,
                  sensorActive := #sensorActive[31],
                  sensorRequested := #sensorRequested[31],
                  sensorMask := #sensorMask[31],
                  sensorStatus => #sensorStatus[31]);
END_REGION
END_FUNCTION

FUNCTION "dintToBool" : Void   // FC10, LAD
{ S7_Optimized_Access := 'TRUE' }
VERSION : 0.1
// stored: AutoNumber true, IsIECCheckEnabled false, SetENOAutomatically false, UDAEnableTagReadback false
BEGIN

REGION Network 1: A INPUTS STATUS
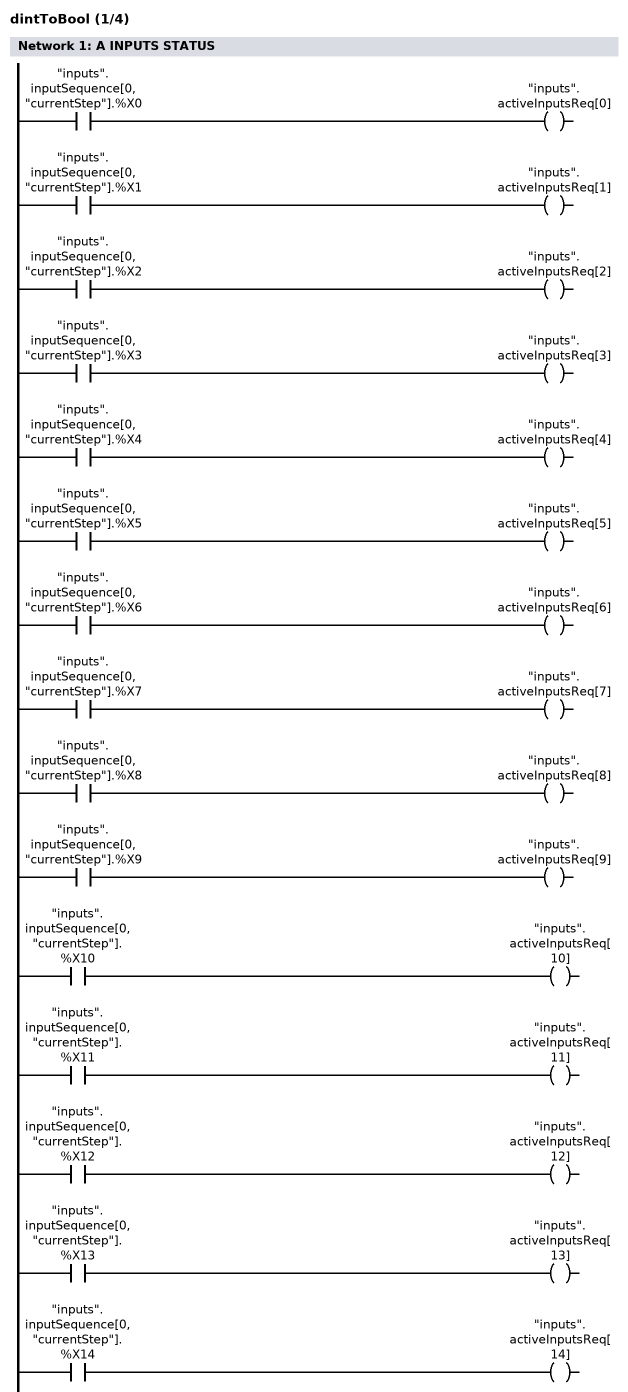
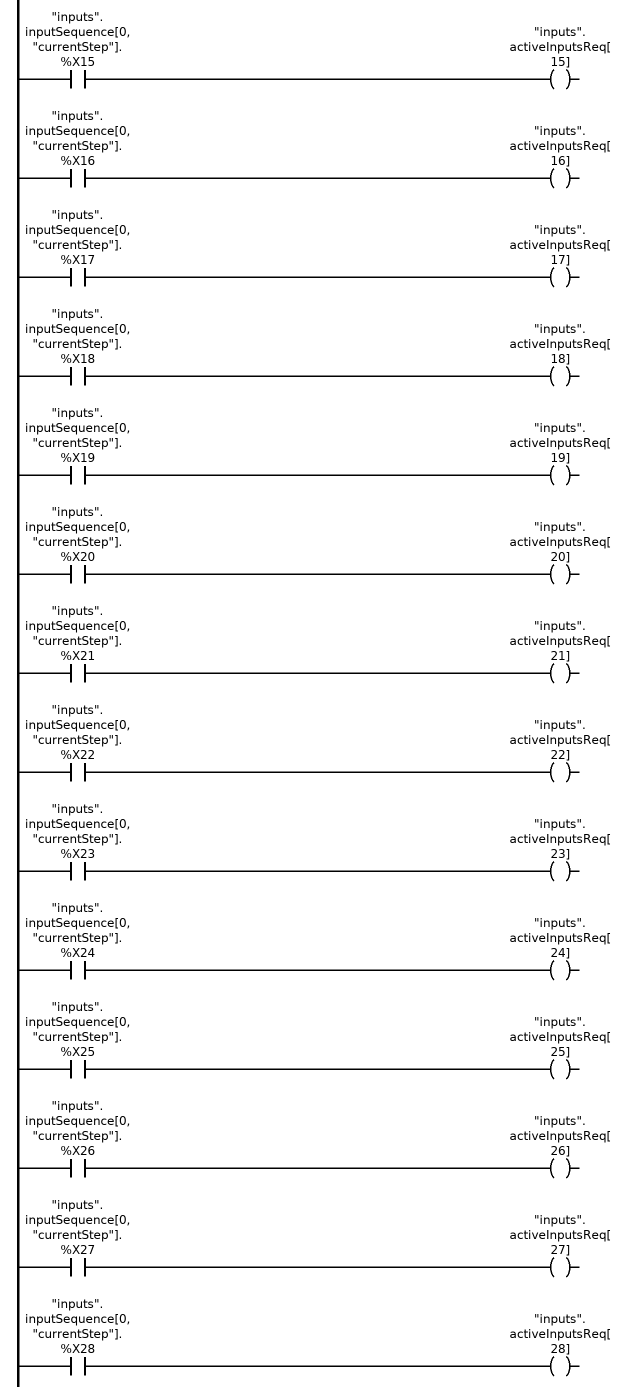
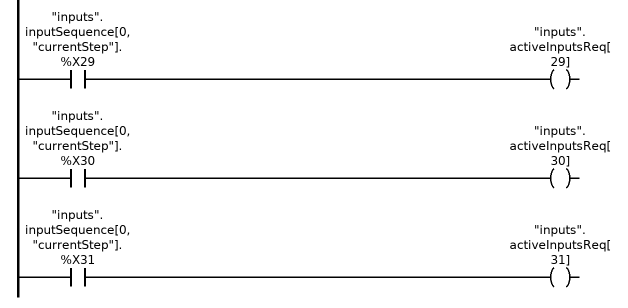
   RUNG wire#powerrail
      Contact( "inputs".inputSequence[0, "currentStep"].%X0 )
      Coil( "inputs".activeInputsReq[0] )
   END_RUNG
   RUNG wire#powerrail
      Contact( "inputs".inputSequence[0, "currentStep"].%X1 )
      Coil( "inputs".activeInputsReq[1] )
   END_RUNG
   RUNG wire#powerrail
      Contact( "inputs".inputSequence[0, "currentStep"].%X2 )
      Coil( "inputs".activeInputsReq[2] )
   END_RUNG
   RUNG wire#powerrail
      Contact( "inputs".inputSequence[0, "currentStep"].%X3 )
      Coil( "inputs".activeInputsReq[3] )
   END_RUNG
   RUNG wire#powerrail
      Contact( "inputs".inputSequence[0, "currentStep"].%X4 )
      Coil( "inputs".activeInputsReq[4] )
   END_RUNG
   RUNG wire#powerrail
      Contact( "inputs".inputSequence[0, "currentStep"].%X5 )
      Coil( "inputs".activeInputsReq[5] )
   END_RUNG
   RUNG wire#powerrail
      Contact( "inputs".inputSequence[0, "currentStep"].%X6 )
      Coil( "inputs".activeInputsReq[6] )
   END_RUNG
   RUNG wire#powerrail
      Contact( "inputs".inputSequence[0, "currentStep"].%X7 )
      Coil( "inputs".activeInputsReq[7] )
   END_RUNG
   RUNG wire#powerrail
      Contact( "inputs".inputSequence[0, "currentStep"].%X8 )
      Coil( "inputs".activeInputsReq[8] )
   END_RUNG
   RUNG wire#powerrail
      Contact( "inputs".inputSequence[0, "currentStep"].%X9 )
      Coil( "inputs".activeInputsReq[9] )
   END_RUNG
   RUNG wire#powerrail
      Contact( "inputs".inputSequence[0, "currentStep"].%X10 )
      Coil( "inputs".activeInputsReq[10] )
   END_RUNG
   RUNG wire#powerrail
      Contact( "inputs".inputSequence[0, "currentStep"].%X11 )
      Coil( "inputs".activeInputsReq[11] )
   END_RUNG
   RUNG wire#powerrail
      Contact( "inputs".inputSequence[0, "currentStep"].%X12 )
      Coil( "inputs".activeInputsReq[12] )
   END_RUNG
   RUNG wire#powerrail
      Contact( "inputs".inputSequence[0, "currentStep"].%X13 )
      Coil( "inputs".activeInputsReq[13] )
   END_RUNG
   RUNG wire#powerrail
      Contact( "inputs".inputSequence[0, "currentStep"].%X14 )
      Coil( "inputs".activeInputsReq[14] )
   END_RUNG
   RUNG wire#powerrail
      Contact( "inputs".inputSequence[0, "currentStep"].%X15 )
      Coil( "inputs".activeInputsReq[15] )
   END_RUNG
   RUNG wire#powerrail
      Contact( "inputs".inputSequence[0, "currentStep"].%X16 )
      Coil( "inputs".activeInputsReq[16] )
   END_RUNG
   RUNG wire#powerrail
      Contact( "inputs".inputSequence[0, "currentStep"].%X17 )
      Coil( "inputs".activeInputsReq[17] )
   END_RUNG
   RUNG wire#powerrail
      Contact( "inputs".inputSequence[0, "currentStep"].%X18 )
      Coil( "inputs".activeInputsReq[18] )
   END_RUNG
   RUNG wire#powerrail
      Contact( "inputs".inputSequence[0, "currentStep"].%X19 )
      Coil( "inputs".activeInputsReq[19] )
   END_RUNG
   RUNG wire#powerrail
      Contact( "inputs".inputSequence[0, "currentStep"].%X20 )
      Coil( "inputs".activeInputsReq[20] )
   END_RUNG
   RUNG wire#powerrail
      Contact( "inputs".inputSequence[0, "currentStep"].%X21 )
      Coil( "inputs".activeInputsReq[21] )
   END_RUNG
   RUNG wire#powerrail
      Contact( "inputs".inputSequence[0, "currentStep"].%X22 )
      Coil( "inputs".activeInputsReq[22] )
   END_RUNG
   RUNG wire#powerrail
      Contact( "inputs".inputSequence[0, "currentStep"].%X23 )
      Coil( "inputs".activeInputsReq[23] )
   END_RUNG
   RUNG wire#powerrail
      Contact( "inputs".inputSequence[0, "currentStep"].%X24 )
      Coil( "inputs".activeInputsReq[24] )
   END_RUNG
   RUNG wire#powerrail
      Contact( "inputs".inputSequence[0, "currentStep"].%X25 )
      Coil( "inputs".activeInputsReq[25] )
   END_RUNG
   RUNG wire#powerrail
      Contact( "inputs".inputSequence[0, "currentStep"].%X26 )
      Coil( "inputs".activeInputsReq[26] )
   END_RUNG
   RUNG wire#powerrail
      Contact( "inputs".inputSequence[0, "currentStep"].%X27 )
      Coil( "inputs".activeInputsReq[27] )
   END_RUNG
   RUNG wire#powerrail
      Contact( "inputs".inputSequence[0, "currentStep"].%X28 )
      Coil( "inputs".activeInputsReq[28] )
   END_RUNG
   RUNG wire#powerrail
      Contact( "inputs".inputSequence[0, "currentStep"].%X29 )
      Coil( "inputs".activeInputsReq[29] )
   END_RUNG
   RUNG wire#powerrail
      Contact( "inputs".inputSequence[0, "currentStep"].%X30 )
      Coil( "inputs".activeInputsReq[30] )
   END_RUNG
   RUNG wire#powerrail
      Contact( "inputs".inputSequence[0, "currentStep"].%X31 )
      Coil( "inputs".activeInputsReq[31] )
   END_RUNG
   // the same network as SCL:
   "inputs".activeInputsReq[0] := "inputs".inputSequence[0, "currentStep"].%X0;
   "inputs".activeInputsReq[1] := "inputs".inputSequence[0, "currentStep"].%X1;
   "inputs".activeInputsReq[2] := "inputs".inputSequence[0, "currentStep"].%X2;
   "inputs".activeInputsReq[3] := "inputs".inputSequence[0, "currentStep"].%X3;
   "inputs".activeInputsReq[4] := "inputs".inputSequence[0, "currentStep"].%X4;
   "inputs".activeInputsReq[5] := "inputs".inputSequence[0, "currentStep"].%X5;
   "inputs".activeInputsReq[6] := "inputs".inputSequence[0, "currentStep"].%X6;
   "inputs".activeInputsReq[7] := "inputs".inputSequence[0, "currentStep"].%X7;
   "inputs".activeInputsReq[8] := "inputs".inputSequence[0, "currentStep"].%X8;
   "inputs".activeInputsReq[9] := "inputs".inputSequence[0, "currentStep"].%X9;
   "inputs".activeInputsReq[10] := "inputs".inputSequence[0, "currentStep"].%X10;
   "inputs".activeInputsReq[11] := "inputs".inputSequence[0, "currentStep"].%X11;
   "inputs".activeInputsReq[12] := "inputs".inputSequence[0, "currentStep"].%X12;
   "inputs".activeInputsReq[13] := "inputs".inputSequence[0, "currentStep"].%X13;
   "inputs".activeInputsReq[14] := "inputs".inputSequence[0, "currentStep"].%X14;
   "inputs".activeInputsReq[15] := "inputs".inputSequence[0, "currentStep"].%X15;
   "inputs".activeInputsReq[16] := "inputs".inputSequence[0, "currentStep"].%X16;
   "inputs".activeInputsReq[17] := "inputs".inputSequence[0, "currentStep"].%X17;
   "inputs".activeInputsReq[18] := "inputs".inputSequence[0, "currentStep"].%X18;
   "inputs".activeInputsReq[19] := "inputs".inputSequence[0, "currentStep"].%X19;
   "inputs".activeInputsReq[20] := "inputs".inputSequence[0, "currentStep"].%X20;
   "inputs".activeInputsReq[21] := "inputs".inputSequence[0, "currentStep"].%X21;
   "inputs".activeInputsReq[22] := "inputs".inputSequence[0, "currentStep"].%X22;
   "inputs".activeInputsReq[23] := "inputs".inputSequence[0, "currentStep"].%X23;
   "inputs".activeInputsReq[24] := "inputs".inputSequence[0, "currentStep"].%X24;
   "inputs".activeInputsReq[25] := "inputs".inputSequence[0, "currentStep"].%X25;
   "inputs".activeInputsReq[26] := "inputs".inputSequence[0, "currentStep"].%X26;
   "inputs".activeInputsReq[27] := "inputs".inputSequence[0, "currentStep"].%X27;
   "inputs".activeInputsReq[28] := "inputs".inputSequence[0, "currentStep"].%X28;
   "inputs".activeInputsReq[29] := "inputs".inputSequence[0, "currentStep"].%X29;
   "inputs".activeInputsReq[30] := "inputs".inputSequence[0, "currentStep"].%X30;
   "inputs".activeInputsReq[31] := "inputs".inputSequence[0, "currentStep"].%X31;
END_REGION

REGION Network 2: MASK INPUTS STATUS
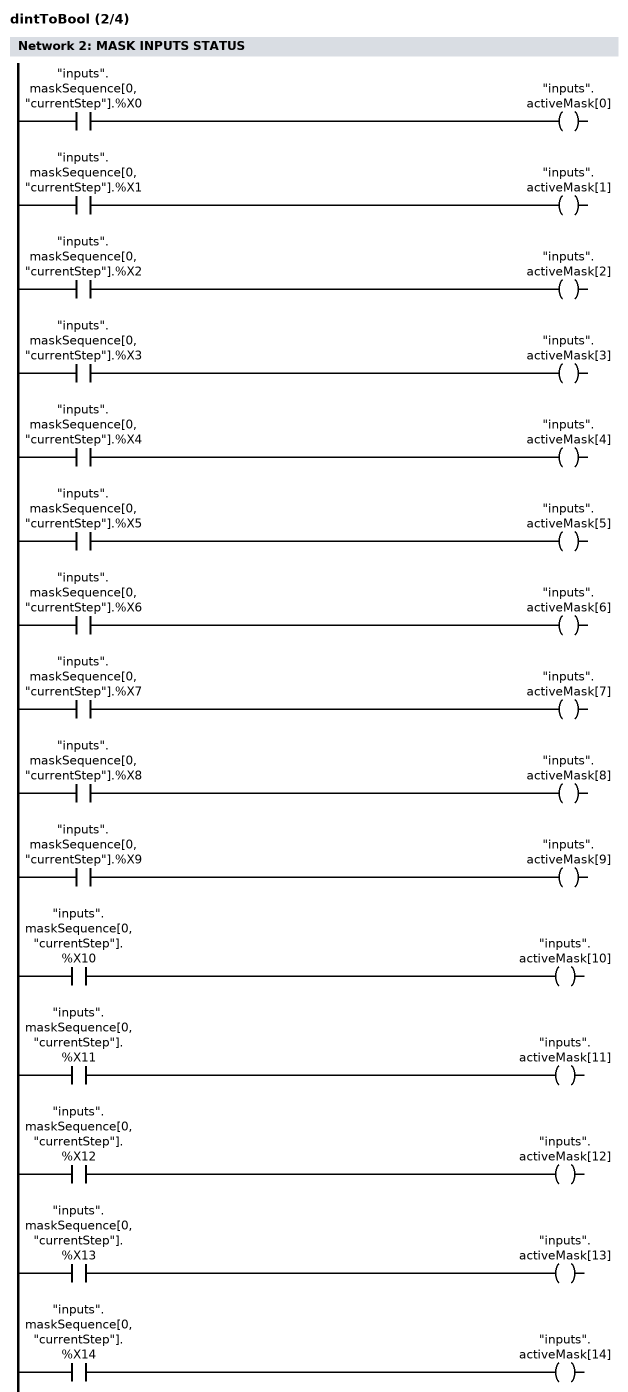
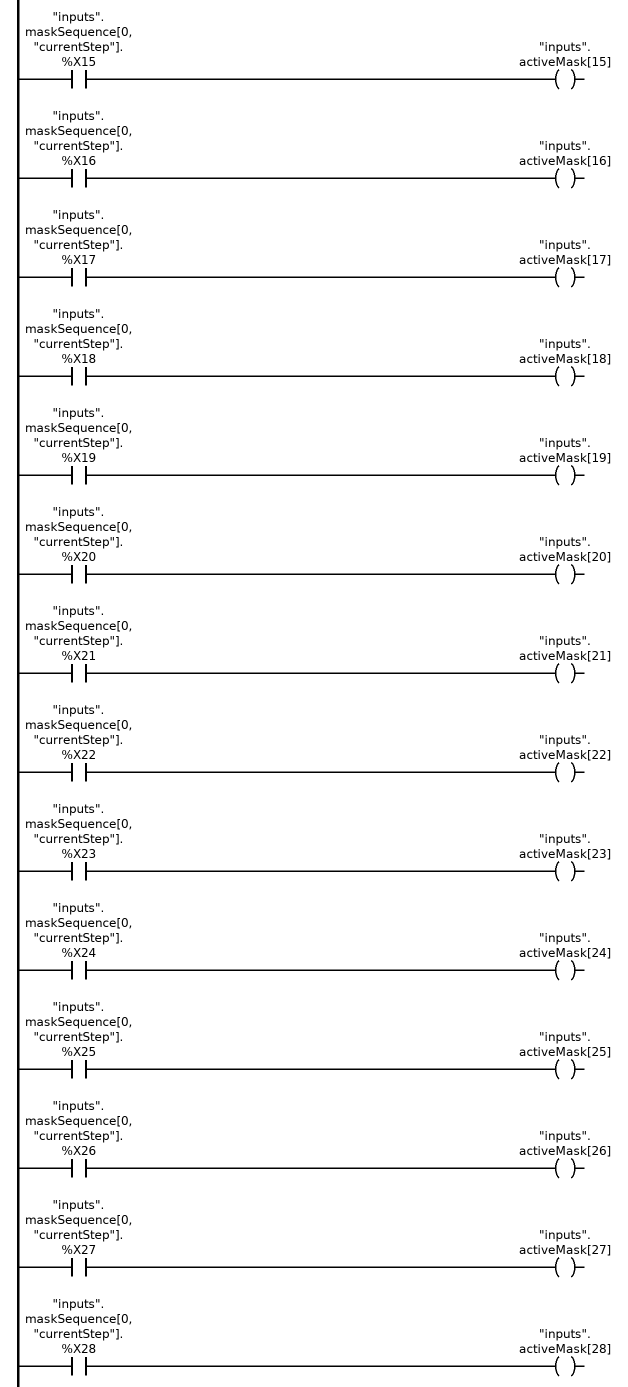
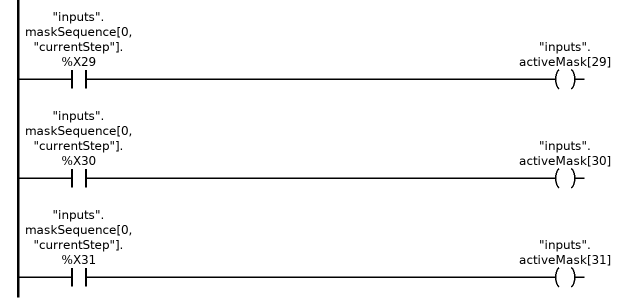
   RUNG wire#powerrail
      Contact( "inputs".maskSequence[0, "currentStep"].%X0 )
      Coil( "inputs".activeMask[0] )
   END_RUNG
   RUNG wire#powerrail
      Contact( "inputs".maskSequence[0, "currentStep"].%X1 )
      Coil( "inputs".activeMask[1] )
   END_RUNG
   RUNG wire#powerrail
      Contact( "inputs".maskSequence[0, "currentStep"].%X2 )
      Coil( "inputs".activeMask[2] )
   END_RUNG
   RUNG wire#powerrail
      Contact( "inputs".maskSequence[0, "currentStep"].%X3 )
      Coil( "inputs".activeMask[3] )
   END_RUNG
   RUNG wire#powerrail
      Contact( "inputs".maskSequence[0, "currentStep"].%X4 )
      Coil( "inputs".activeMask[4] )
   END_RUNG
   RUNG wire#powerrail
      Contact( "inputs".maskSequence[0, "currentStep"].%X5 )
      Coil( "inputs".activeMask[5] )
   END_RUNG
   RUNG wire#powerrail
      Contact( "inputs".maskSequence[0, "currentStep"].%X6 )
      Coil( "inputs".activeMask[6] )
   END_RUNG
   RUNG wire#powerrail
      Contact( "inputs".maskSequence[0, "currentStep"].%X7 )
      Coil( "inputs".activeMask[7] )
   END_RUNG
   RUNG wire#powerrail
      Contact( "inputs".maskSequence[0, "currentStep"].%X8 )
      Coil( "inputs".activeMask[8] )
   END_RUNG
   RUNG wire#powerrail
      Contact( "inputs".maskSequence[0, "currentStep"].%X9 )
      Coil( "inputs".activeMask[9] )
   END_RUNG
   RUNG wire#powerrail
      Contact( "inputs".maskSequence[0, "currentStep"].%X10 )
      Coil( "inputs".activeMask[10] )
   END_RUNG
   RUNG wire#powerrail
      Contact( "inputs".maskSequence[0, "currentStep"].%X11 )
      Coil( "inputs".activeMask[11] )
   END_RUNG
   RUNG wire#powerrail
      Contact( "inputs".maskSequence[0, "currentStep"].%X12 )
      Coil( "inputs".activeMask[12] )
   END_RUNG
   RUNG wire#powerrail
      Contact( "inputs".maskSequence[0, "currentStep"].%X13 )
      Coil( "inputs".activeMask[13] )
   END_RUNG
   RUNG wire#powerrail
      Contact( "inputs".maskSequence[0, "currentStep"].%X14 )
      Coil( "inputs".activeMask[14] )
   END_RUNG
   RUNG wire#powerrail
      Contact( "inputs".maskSequence[0, "currentStep"].%X15 )
      Coil( "inputs".activeMask[15] )
   END_RUNG
   RUNG wire#powerrail
      Contact( "inputs".maskSequence[0, "currentStep"].%X16 )
      Coil( "inputs".activeMask[16] )
   END_RUNG
   RUNG wire#powerrail
      Contact( "inputs".maskSequence[0, "currentStep"].%X17 )
      Coil( "inputs".activeMask[17] )
   END_RUNG
   RUNG wire#powerrail
      Contact( "inputs".maskSequence[0, "currentStep"].%X18 )
      Coil( "inputs".activeMask[18] )
   END_RUNG
   RUNG wire#powerrail
      Contact( "inputs".maskSequence[0, "currentStep"].%X19 )
      Coil( "inputs".activeMask[19] )
   END_RUNG
   RUNG wire#powerrail
      Contact( "inputs".maskSequence[0, "currentStep"].%X20 )
      Coil( "inputs".activeMask[20] )
   END_RUNG
   RUNG wire#powerrail
      Contact( "inputs".maskSequence[0, "currentStep"].%X21 )
      Coil( "inputs".activeMask[21] )
   END_RUNG
   RUNG wire#powerrail
      Contact( "inputs".maskSequence[0, "currentStep"].%X22 )
      Coil( "inputs".activeMask[22] )
   END_RUNG
   RUNG wire#powerrail
      Contact( "inputs".maskSequence[0, "currentStep"].%X23 )
      Coil( "inputs".activeMask[23] )
   END_RUNG
   RUNG wire#powerrail
      Contact( "inputs".maskSequence[0, "currentStep"].%X24 )
      Coil( "inputs".activeMask[24] )
   END_RUNG
   RUNG wire#powerrail
      Contact( "inputs".maskSequence[0, "currentStep"].%X25 )
      Coil( "inputs".activeMask[25] )
   END_RUNG
   RUNG wire#powerrail
      Contact( "inputs".maskSequence[0, "currentStep"].%X26 )
      Coil( "inputs".activeMask[26] )
   END_RUNG
   RUNG wire#powerrail
      Contact( "inputs".maskSequence[0, "currentStep"].%X27 )
      Coil( "inputs".activeMask[27] )
   END_RUNG
   RUNG wire#powerrail
      Contact( "inputs".maskSequence[0, "currentStep"].%X28 )
      Coil( "inputs".activeMask[28] )
   END_RUNG
   RUNG wire#powerrail
      Contact( "inputs".maskSequence[0, "currentStep"].%X29 )
      Coil( "inputs".activeMask[29] )
   END_RUNG
   RUNG wire#powerrail
      Contact( "inputs".maskSequence[0, "currentStep"].%X30 )
      Coil( "inputs".activeMask[30] )
   END_RUNG
   RUNG wire#powerrail
      Contact( "inputs".maskSequence[0, "currentStep"].%X31 )
      Coil( "inputs".activeMask[31] )
   END_RUNG
   // the same network as SCL:
   "inputs".activeMask[0] := "inputs".maskSequence[0, "currentStep"].%X0;
   "inputs".activeMask[1] := "inputs".maskSequence[0, "currentStep"].%X1;
   "inputs".activeMask[2] := "inputs".maskSequence[0, "currentStep"].%X2;
   "inputs".activeMask[3] := "inputs".maskSequence[0, "currentStep"].%X3;
   "inputs".activeMask[4] := "inputs".maskSequence[0, "currentStep"].%X4;
   "inputs".activeMask[5] := "inputs".maskSequence[0, "currentStep"].%X5;
   "inputs".activeMask[6] := "inputs".maskSequence[0, "currentStep"].%X6;
   "inputs".activeMask[7] := "inputs".maskSequence[0, "currentStep"].%X7;
   "inputs".activeMask[8] := "inputs".maskSequence[0, "currentStep"].%X8;
   "inputs".activeMask[9] := "inputs".maskSequence[0, "currentStep"].%X9;
   "inputs".activeMask[10] := "inputs".maskSequence[0, "currentStep"].%X10;
   "inputs".activeMask[11] := "inputs".maskSequence[0, "currentStep"].%X11;
   "inputs".activeMask[12] := "inputs".maskSequence[0, "currentStep"].%X12;
   "inputs".activeMask[13] := "inputs".maskSequence[0, "currentStep"].%X13;
   "inputs".activeMask[14] := "inputs".maskSequence[0, "currentStep"].%X14;
   "inputs".activeMask[15] := "inputs".maskSequence[0, "currentStep"].%X15;
   "inputs".activeMask[16] := "inputs".maskSequence[0, "currentStep"].%X16;
   "inputs".activeMask[17] := "inputs".maskSequence[0, "currentStep"].%X17;
   "inputs".activeMask[18] := "inputs".maskSequence[0, "currentStep"].%X18;
   "inputs".activeMask[19] := "inputs".maskSequence[0, "currentStep"].%X19;
   "inputs".activeMask[20] := "inputs".maskSequence[0, "currentStep"].%X20;
   "inputs".activeMask[21] := "inputs".maskSequence[0, "currentStep"].%X21;
   "inputs".activeMask[22] := "inputs".maskSequence[0, "currentStep"].%X22;
   "inputs".activeMask[23] := "inputs".maskSequence[0, "currentStep"].%X23;
   "inputs".activeMask[24] := "inputs".maskSequence[0, "currentStep"].%X24;
   "inputs".activeMask[25] := "inputs".maskSequence[0, "currentStep"].%X25;
   "inputs".activeMask[26] := "inputs".maskSequence[0, "currentStep"].%X26;
   "inputs".activeMask[27] := "inputs".maskSequence[0, "currentStep"].%X27;
   "inputs".activeMask[28] := "inputs".maskSequence[0, "currentStep"].%X28;
   "inputs".activeMask[29] := "inputs".maskSequence[0, "currentStep"].%X29;
   "inputs".activeMask[30] := "inputs".maskSequence[0, "currentStep"].%X30;
   "inputs".activeMask[31] := "inputs".maskSequence[0, "currentStep"].%X31;
END_REGION

REGION Network 3: B OUTPUTS STATUS
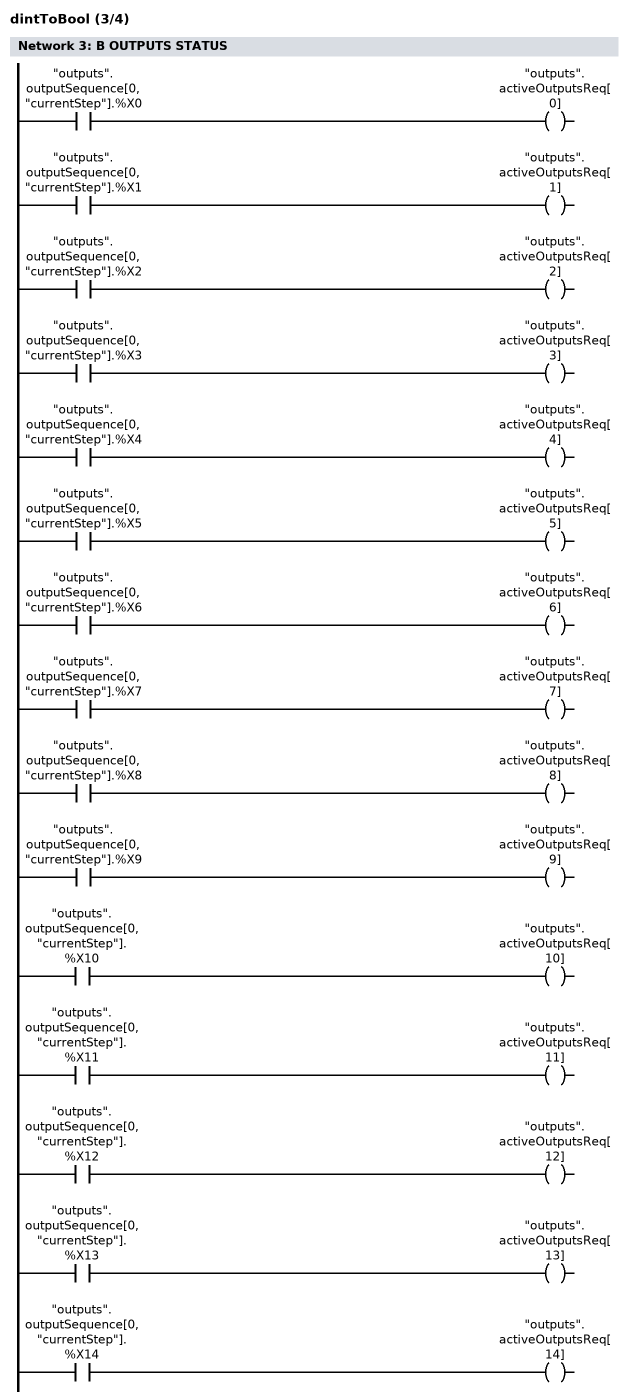
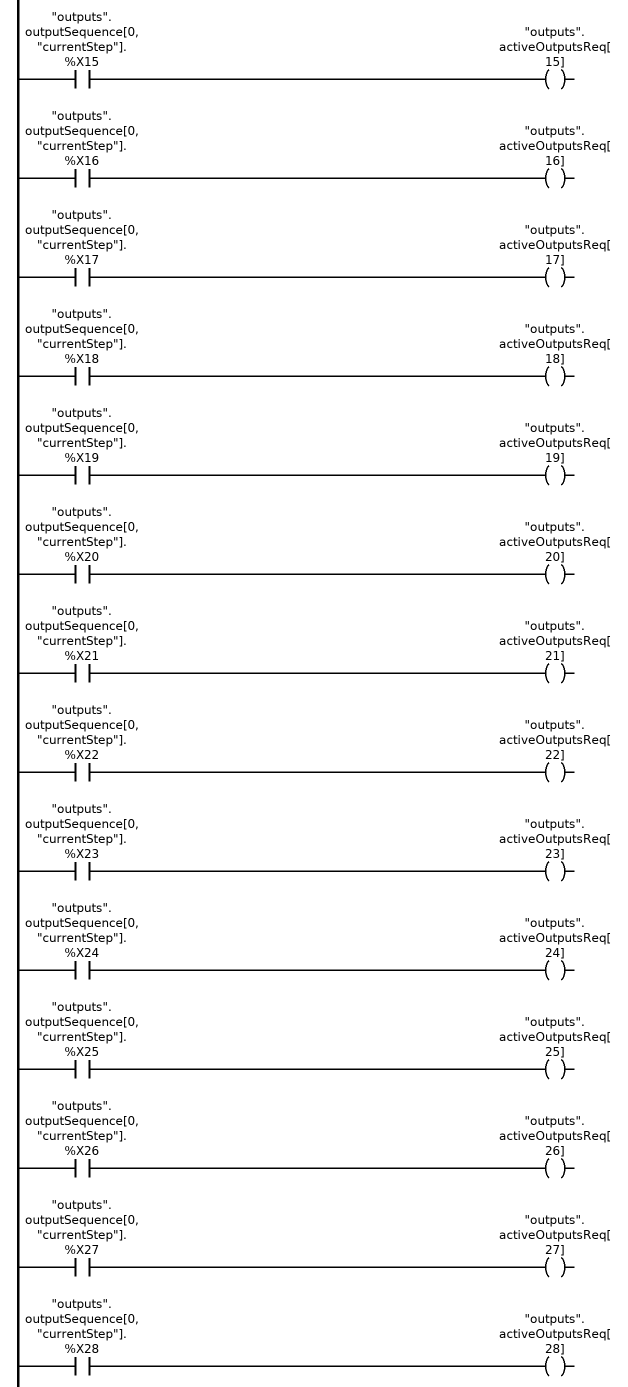
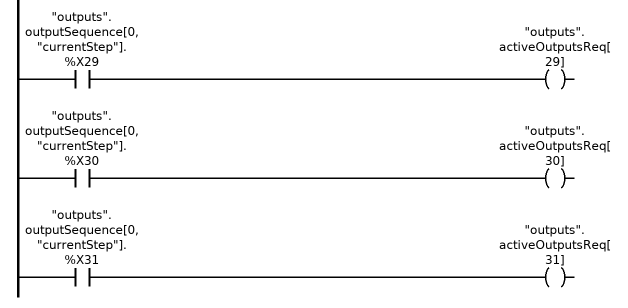
   RUNG wire#powerrail
      Contact( "outputs".outputSequence[0, "currentStep"].%X0 )
      Coil( "outputs".activeOutputsReq[0] )
   END_RUNG
   RUNG wire#powerrail
      Contact( "outputs".outputSequence[0, "currentStep"].%X1 )
      Coil( "outputs".activeOutputsReq[1] )
   END_RUNG
   RUNG wire#powerrail
      Contact( "outputs".outputSequence[0, "currentStep"].%X2 )
      Coil( "outputs".activeOutputsReq[2] )
   END_RUNG
   RUNG wire#powerrail
      Contact( "outputs".outputSequence[0, "currentStep"].%X3 )
      Coil( "outputs".activeOutputsReq[3] )
   END_RUNG
   RUNG wire#powerrail
      Contact( "outputs".outputSequence[0, "currentStep"].%X4 )
      Coil( "outputs".activeOutputsReq[4] )
   END_RUNG
   RUNG wire#powerrail
      Contact( "outputs".outputSequence[0, "currentStep"].%X5 )
      Coil( "outputs".activeOutputsReq[5] )
   END_RUNG
   RUNG wire#powerrail
      Contact( "outputs".outputSequence[0, "currentStep"].%X6 )
      Coil( "outputs".activeOutputsReq[6] )
   END_RUNG
   RUNG wire#powerrail
      Contact( "outputs".outputSequence[0, "currentStep"].%X7 )
      Coil( "outputs".activeOutputsReq[7] )
   END_RUNG
   RUNG wire#powerrail
      Contact( "outputs".outputSequence[0, "currentStep"].%X8 )
      Coil( "outputs".activeOutputsReq[8] )
   END_RUNG
   RUNG wire#powerrail
      Contact( "outputs".outputSequence[0, "currentStep"].%X9 )
      Coil( "outputs".activeOutputsReq[9] )
   END_RUNG
   RUNG wire#powerrail
      Contact( "outputs".outputSequence[0, "currentStep"].%X10 )
      Coil( "outputs".activeOutputsReq[10] )
   END_RUNG
   RUNG wire#powerrail
      Contact( "outputs".outputSequence[0, "currentStep"].%X11 )
      Coil( "outputs".activeOutputsReq[11] )
   END_RUNG
   RUNG wire#powerrail
      Contact( "outputs".outputSequence[0, "currentStep"].%X12 )
      Coil( "outputs".activeOutputsReq[12] )
   END_RUNG
   RUNG wire#powerrail
      Contact( "outputs".outputSequence[0, "currentStep"].%X13 )
      Coil( "outputs".activeOutputsReq[13] )
   END_RUNG
   RUNG wire#powerrail
      Contact( "outputs".outputSequence[0, "currentStep"].%X14 )
      Coil( "outputs".activeOutputsReq[14] )
   END_RUNG
   RUNG wire#powerrail
      Contact( "outputs".outputSequence[0, "currentStep"].%X15 )
      Coil( "outputs".activeOutputsReq[15] )
   END_RUNG
   RUNG wire#powerrail
      Contact( "outputs".outputSequence[0, "currentStep"].%X16 )
      Coil( "outputs".activeOutputsReq[16] )
   END_RUNG
   RUNG wire#powerrail
      Contact( "outputs".outputSequence[0, "currentStep"].%X17 )
      Coil( "outputs".activeOutputsReq[17] )
   END_RUNG
   RUNG wire#powerrail
      Contact( "outputs".outputSequence[0, "currentStep"].%X18 )
      Coil( "outputs".activeOutputsReq[18] )
   END_RUNG
   RUNG wire#powerrail
      Contact( "outputs".outputSequence[0, "currentStep"].%X19 )
      Coil( "outputs".activeOutputsReq[19] )
   END_RUNG
   RUNG wire#powerrail
      Contact( "outputs".outputSequence[0, "currentStep"].%X20 )
      Coil( "outputs".activeOutputsReq[20] )
   END_RUNG
   RUNG wire#powerrail
      Contact( "outputs".outputSequence[0, "currentStep"].%X21 )
      Coil( "outputs".activeOutputsReq[21] )
   END_RUNG
   RUNG wire#powerrail
      Contact( "outputs".outputSequence[0, "currentStep"].%X22 )
      Coil( "outputs".activeOutputsReq[22] )
   END_RUNG
   RUNG wire#powerrail
      Contact( "outputs".outputSequence[0, "currentStep"].%X23 )
      Coil( "outputs".activeOutputsReq[23] )
   END_RUNG
   RUNG wire#powerrail
      Contact( "outputs".outputSequence[0, "currentStep"].%X24 )
      Coil( "outputs".activeOutputsReq[24] )
   END_RUNG
   RUNG wire#powerrail
      Contact( "outputs".outputSequence[0, "currentStep"].%X25 )
      Coil( "outputs".activeOutputsReq[25] )
   END_RUNG
   RUNG wire#powerrail
      Contact( "outputs".outputSequence[0, "currentStep"].%X26 )
      Coil( "outputs".activeOutputsReq[26] )
   END_RUNG
   RUNG wire#powerrail
      Contact( "outputs".outputSequence[0, "currentStep"].%X27 )
      Coil( "outputs".activeOutputsReq[27] )
   END_RUNG
   RUNG wire#powerrail
      Contact( "outputs".outputSequence[0, "currentStep"].%X28 )
      Coil( "outputs".activeOutputsReq[28] )
   END_RUNG
   RUNG wire#powerrail
      Contact( "outputs".outputSequence[0, "currentStep"].%X29 )
      Coil( "outputs".activeOutputsReq[29] )
   END_RUNG
   RUNG wire#powerrail
      Contact( "outputs".outputSequence[0, "currentStep"].%X30 )
      Coil( "outputs".activeOutputsReq[30] )
   END_RUNG
   RUNG wire#powerrail
      Contact( "outputs".outputSequence[0, "currentStep"].%X31 )
      Coil( "outputs".activeOutputsReq[31] )
   END_RUNG
   // the same network as SCL:
   "outputs".activeOutputsReq[0] := "outputs".outputSequence[0, "currentStep"].%X0;
   "outputs".activeOutputsReq[1] := "outputs".outputSequence[0, "currentStep"].%X1;
   "outputs".activeOutputsReq[2] := "outputs".outputSequence[0, "currentStep"].%X2;
   "outputs".activeOutputsReq[3] := "outputs".outputSequence[0, "currentStep"].%X3;
   "outputs".activeOutputsReq[4] := "outputs".outputSequence[0, "currentStep"].%X4;
   "outputs".activeOutputsReq[5] := "outputs".outputSequence[0, "currentStep"].%X5;
   "outputs".activeOutputsReq[6] := "outputs".outputSequence[0, "currentStep"].%X6;
   "outputs".activeOutputsReq[7] := "outputs".outputSequence[0, "currentStep"].%X7;
   "outputs".activeOutputsReq[8] := "outputs".outputSequence[0, "currentStep"].%X8;
   "outputs".activeOutputsReq[9] := "outputs".outputSequence[0, "currentStep"].%X9;
   "outputs".activeOutputsReq[10] := "outputs".outputSequence[0, "currentStep"].%X10;
   "outputs".activeOutputsReq[11] := "outputs".outputSequence[0, "currentStep"].%X11;
   "outputs".activeOutputsReq[12] := "outputs".outputSequence[0, "currentStep"].%X12;
   "outputs".activeOutputsReq[13] := "outputs".outputSequence[0, "currentStep"].%X13;
   "outputs".activeOutputsReq[14] := "outputs".outputSequence[0, "currentStep"].%X14;
   "outputs".activeOutputsReq[15] := "outputs".outputSequence[0, "currentStep"].%X15;
   "outputs".activeOutputsReq[16] := "outputs".outputSequence[0, "currentStep"].%X16;
   "outputs".activeOutputsReq[17] := "outputs".outputSequence[0, "currentStep"].%X17;
   "outputs".activeOutputsReq[18] := "outputs".outputSequence[0, "currentStep"].%X18;
   "outputs".activeOutputsReq[19] := "outputs".outputSequence[0, "currentStep"].%X19;
   "outputs".activeOutputsReq[20] := "outputs".outputSequence[0, "currentStep"].%X20;
   "outputs".activeOutputsReq[21] := "outputs".outputSequence[0, "currentStep"].%X21;
   "outputs".activeOutputsReq[22] := "outputs".outputSequence[0, "currentStep"].%X22;
   "outputs".activeOutputsReq[23] := "outputs".outputSequence[0, "currentStep"].%X23;
   "outputs".activeOutputsReq[24] := "outputs".outputSequence[0, "currentStep"].%X24;
   "outputs".activeOutputsReq[25] := "outputs".outputSequence[0, "currentStep"].%X25;
   "outputs".activeOutputsReq[26] := "outputs".outputSequence[0, "currentStep"].%X26;
   "outputs".activeOutputsReq[27] := "outputs".outputSequence[0, "currentStep"].%X27;
   "outputs".activeOutputsReq[28] := "outputs".outputSequence[0, "currentStep"].%X28;
   "outputs".activeOutputsReq[29] := "outputs".outputSequence[0, "currentStep"].%X29;
   "outputs".activeOutputsReq[30] := "outputs".outputSequence[0, "currentStep"].%X30;
   "outputs".activeOutputsReq[31] := "outputs".outputSequence[0, "currentStep"].%X31;
END_REGION

REGION Network 4: MASK OUTPUTS STATUS
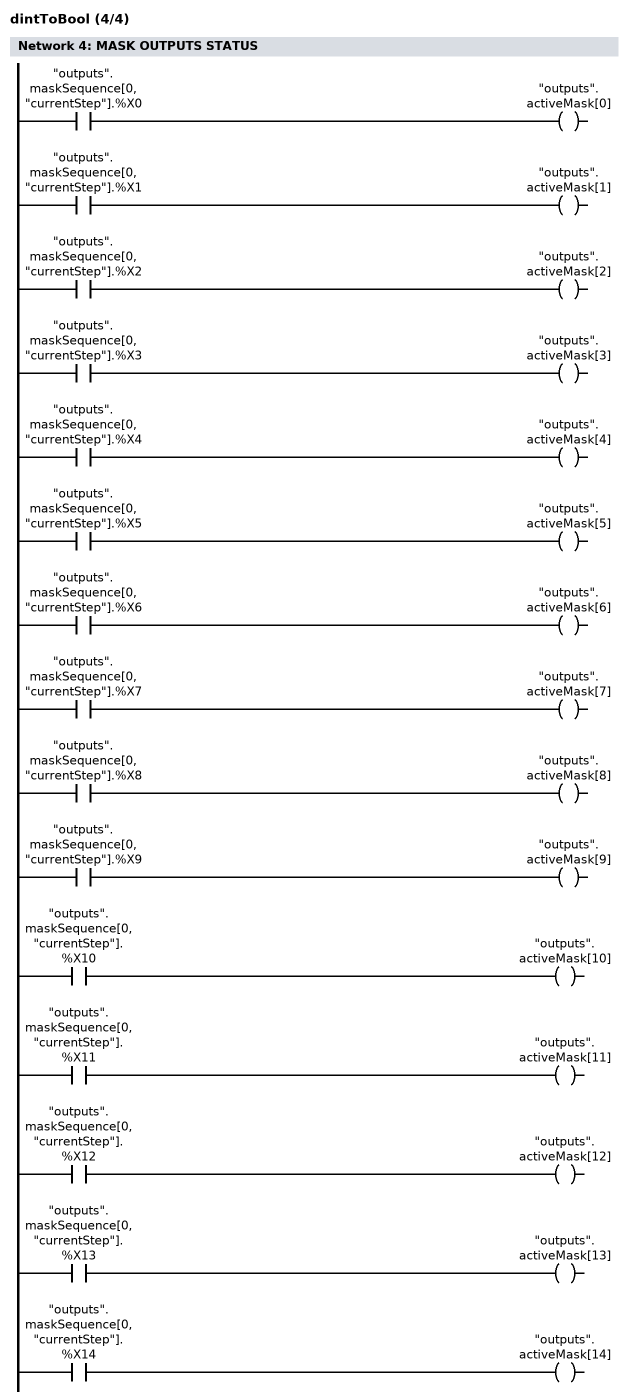
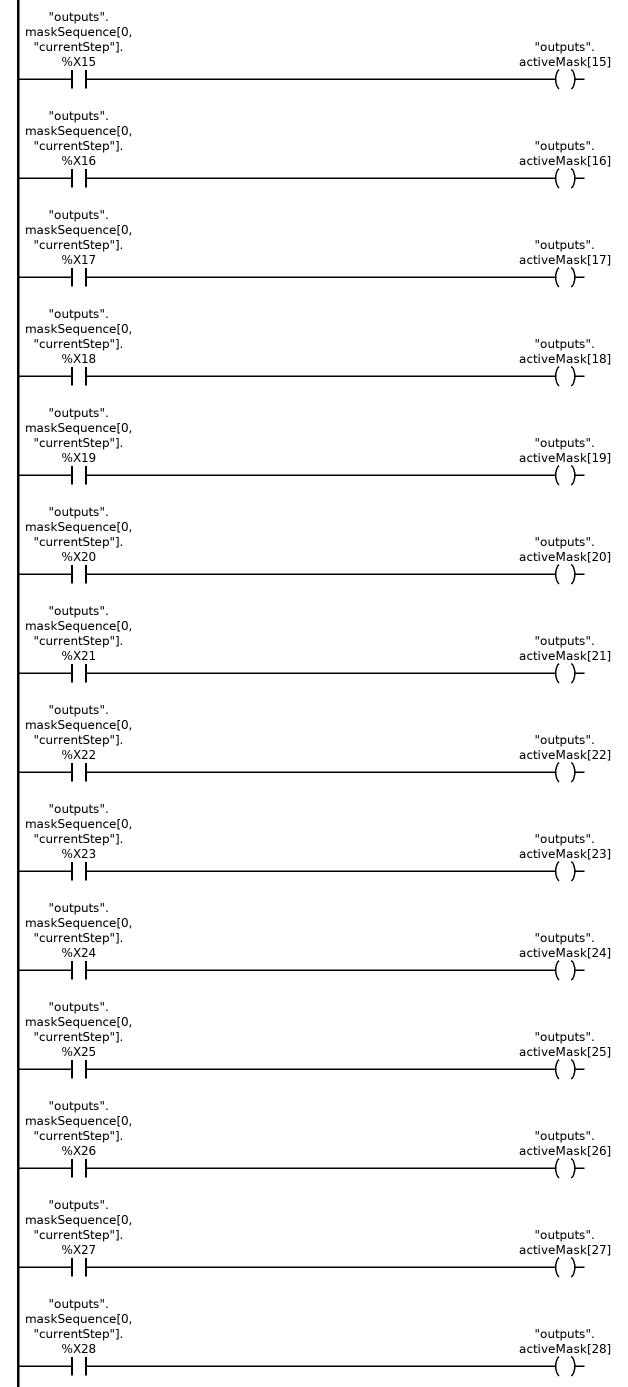
